ptrConfigPage^.aiFTrigActionPanelRight[5]:=0;
ptrConfigPage^.aiRTrigActionFunctionPanel[1]:=0;
ptrConfigPage^.aiRTrigActionFunctionPanel[2]:=0;
ptrConfigPage^.aiRTrigActionFunctionPanel[3]:=0;
ptrConfigPage^.aiRTrigActionFunctionPanel[4]:=0;
ptrConfigPage^.aiRTrigActionFunctionPanel[5]:=0;
ptrConfigPage^.aiRTrigActionFunctionPanel[6]:=0;
ptrConfigPage^.aiRTrigActionFunctionPanel[7]:=0;
ptrConfigPage^.aiRTrigActionFunctionPanel[8]:=0;
ptrConfigPage^.aiRTrigActionFunctionPanel[9]:=0;
ptrConfigPage^.aiRTrigActionFunctionPanel[10]:=0;
ptrConfigPage^.aiRTrigActionFunctionPanel[11]:=0;
ptrConfigPage^.aiRTrigActionFunctionPanel[12]:=0;
TaskBar_SetupModeB;
ptrConfigPage^.xMaskBtStart:=FALSE;
ptrConfigPage^.xMaskBtStop:=TRUE;
END_ACTION
ACTION TaskBar_BIOS:
(* Navigation panel restriction *)
ptrConfigPage^.aiRTrigActionTouchScreenNavPanel[1,1]:=0;
ptrConfigPage^.aiRTrigActionTouchScreenNavPanel[1,2]:=0;
ptrConfigPage^.aiRTrigActionTouchScreenNavPanel[1,3]:=0;
ptrConfigPage^.aiRTrigActionTouchScreenNavPanel[1,4]:=0;
ptrConfigPage^.aiRTrigActionTouchScreenNavPanel[1,5]:=0;
ptrConfigPage^.aiRTrigActionTouchScreenNavPanel[1,6]:=0;
ptrConfigPage^.aiRTrigActionTouchScreenNavPanel[1,7]:=0;
ptrConfigPage^.aiRTrigActionTouchScreenNavPanel[1,8]:=0;
ptrConfigPage^.aiRTrigActionTouchScreenNavPanel[1,9]:=0;
ptrConfigPage^.aiRTrigActionTouchScreenNavPanel[2,1]:=0;
ptrConfigPage^.aiRTrigActionTouchScreenNavPanel[2,2]:=0;
ptrConfigPage^.aiRTrigActionTouchScreenNavPanel[2,3]:=0;
ptrConfigPage^.aiRTrigActionTouchScreenNavPanel[2,4]:=0;
ptrConfigPage^.aiRTrigActionTouchScreenNavPanel[2,5]:=0;
ptrConfigPage^.aiRTrigActionTouchScreenNavPanel[2,6]:=0;
ptrConfigPage^.aiRTrigActionTouchScreenNavPanel[2,7]:=0;
ptrConfigPage^.aiRTrigActionTouchScreenNavPanel[2,8]:=0;
ptrConfigPage^.aiRTrigActionTouchScreenNavPanel[2,9]:=0;
ptrConfigPage^.aiRTrigActionTouchScreenNavPanel[3,1]:=0;
ptrConfigPage^.aiRTrigActionTouchScreenNavPanel[3,2]:=0;
ptrConfigPage^.aiRTrigActionTouchScreenNavPanel[3,3]:=0;
ptrConfigPage^.aiRTrigActionTouchScreenNavPanel[3,4]:=0;
ptrConfigPage^.aiRTrigActionTouchScreenNavPanel[3,5]:=0;
ptrConfigPage^.aiRTrigActionTouchScreenNavPanel[3,6]:=0;
ptrConfigPage^.aiRTrigActionTouchScreenNavPanel[3,7]:=0;
ptrConfigPage^.aiRTrigActionTouchScreenNavPanel[3,8]:=0;
ptrConfigPage^.aiRTrigActionTouchScreenNavPanel[3,9]:=0;
ptrConfigPage^.aiRTrigActionTouchScreenNavPanel[4,1]:=0;
ptrConfigPage^.aiRTrigActionTouchScreenNavPanel[4,2]:=0;
ptrConfigPage^.aiRTrigActionTouchScreenNavPanel[4,3]:=0;
ptrConfigPage^.aiRTrigActionTouchScreenNavPanel[4,4]:=0;
ptrConfigPage^.aiRTrigActionTouchScreenNavPanel[4,5]:=0;
ptrConfigPage^.aiRTrigActionTouchScreenNavPanel[4,6]:=0;
ptrConfigPage^.aiRTrigActionTouchScreenNavPanel[4,7]:=0;
ptrConfigPage^.aiRTrigActionTouchScreenNavPanel[4,8]:=0;
ptrConfigPage^.aiRTrigActionTouchScreenNavPanel[4,9]:=0;
ptrConfigPage^.aiRTrigActionTouchScreenNavPanel[5,1]:=0;
ptrConfigPage^.aiRTrigActionTouchScreenNavPanel[5,2]:=0;
ptrConfigPage^.aiRTrigActionTouchScreenNavPanel[5,3]:=0;
ptrConfigPage^.aiRTrigActionTouchScreenNavPanel[5,4]:=0;
ptrConfigPage^.aiRTrigActionTouchScreenNavPanel[5,5]:=0;
ptrConfigPage^.aiRTrigActionTouchScreenNavPanel[5,6]:=0;
ptrConfigPage^.aiRTrigActionTouchScreenNavPanel[5,7]:=0;
ptrConfigPage^.aiRTrigActionTouchScreenNavPanel[5,8]:=0;
ptrConfigPage^.aiRTrigActionTouchScreenNavPanel[5,9]:=0;
ptrConfigPage^.aiRTrigActionTouchScreenNavPanel[6,1]:=0;
ptrConfigPage^.aiRTrigActionTouchScreenNavPanel[6,2]:=0;
ptrConfigPage^.aiRTrigActionTouchScreenNavPanel[6,3]:=0;
ptrConfigPage^.aiRTrigActionTouchScreenNavPanel[6,4]:=0;
ptrConfigPage^.aiRTrigActionTouchScreenNavPanel[6,5]:=0;
ptrConfigPage^.aiRTrigActionTouchScreenNavPanel[6,6]:=0;
ptrConfigPage^.aiRTrigActionTouchScreenNavPanel[6,7]:=0;
ptrConfigPage^.aiRTrigActionTouchScreenNavPanel[6,8]:=0;
ptrConfigPage^.aiRTrigActionTouchScreenNavPanel[6,9]:=0;
END_ACTION
ACTION TaskBar_NormalMode:
(* Navigation panel restriction *)
ptrConfigPage^.wMaskTouchScreenNavPanel:=16#3F;
ptrConfigPage^.aiRTrigActionTouchScreenNavPanel[1,1]:=10000 + gT_PageNumber.iAutoMode_Process;
ptrConfigPage^.aiRTrigActionTouchScreenNavPanel[1,2]:=10000 + gT_PageNumber.iAutoMode_ProcessValue1;	(* IGS *)
ptrConfigPage^.aiRTrigActionTouchScreenNavPanel[1,3]:=10000 + gT_PageNumber.iAutoMode_ProcessValue2;	(* IGS *)
ptrConfigPage^.aiRTrigActionTouchScreenNavPanel[1,4]:=10000 + gT_PageNumber.iAutoMode_PartQuality;
ptrConfigPage^.aiRTrigActionTouchScreenNavPanel[1,5]:=0;
ptrConfigPage^.aiRTrigActionTouchScreenNavPanel[1,6]:=0;
ptrConfigPage^.aiRTrigActionTouchScreenNavPanel[1,7]:=0;
ptrConfigPage^.aiRTrigActionTouchScreenNavPanel[1,8]:=0;
ptrConfigPage^.aiRTrigActionTouchScreenNavPanel[1,9]:=0;
ptrConfigPage^.aiRTrigActionTouchScreenNavPanel[2,1]:=10000 + gT_PageNumber.iAutoMode_Referencing;
ptrConfigPage^.aiRTrigActionTouchScreenNavPanel[2,2]:=0;
ptrConfigPage^.aiRTrigActionTouchScreenNavPanel[2,3]:=0;
ptrConfigPage^.aiRTrigActionTouchScreenNavPanel[2,4]:=0;
ptrConfigPage^.aiRTrigActionTouchScreenNavPanel[2,5]:=0;
ptrConfigPage^.aiRTrigActionTouchScreenNavPanel[2,6]:=0;
ptrConfigPage^.aiRTrigActionTouchScreenNavPanel[2,7]:=0;
ptrConfigPage^.aiRTrigActionTouchScreenNavPanel[2,8]:=0;
ptrConfigPage^.aiRTrigActionTouchScreenNavPanel[2,9]:=0;
ptrConfigPage^.aiRTrigActionTouchScreenNavPanel[3,1]:=10000 + gT_PageNumber.iAutoMode_Profile;
ptrConfigPage^.aiRTrigActionTouchScreenNavPanel[3,2]:=0;
ptrConfigPage^.aiRTrigActionTouchScreenNavPanel[3,3]:=0;
ptrConfigPage^.aiRTrigActionTouchScreenNavPanel[3,4]:=0;
ptrConfigPage^.aiRTrigActionTouchScreenNavPanel[3,5]:=0;
ptrConfigPage^.aiRTrigActionTouchScreenNavPanel[3,6]:=0;
ptrConfigPage^.aiRTrigActionTouchScreenNavPanel[3,7]:=0;
ptrConfigPage^.aiRTrigActionTouchScreenNavPanel[3,8]:=0;
ptrConfigPage^.aiRTrigActionTouchScreenNavPanel[3,9]:=0;
ptrConfigPage^.aiRTrigActionTouchScreenNavPanel[4,1]:=10000 + gT_PageNumber.iAutoMode_ToolChange;
ptrConfigPage^.aiRTrigActionTouchScreenNavPanel[4,2]:=10000 + gT_PageNumber.iAutoMode_UserLevel;
ptrConfigPage^.aiRTrigActionTouchScreenNavPanel[4,3]:=10000 + gT_PageNumber.iAutoMode_Language;
ptrConfigPage^.aiRTrigActionTouchScreenNavPanel[4,4]:=0;
ptrConfigPage^.aiRTrigActionTouchScreenNavPanel[4,5]:=0;
ptrConfigPage^.aiRTrigActionTouchScreenNavPanel[4,6]:=0;
ptrConfigPage^.aiRTrigActionTouchScreenNavPanel[4,7]:=0;
ptrConfigPage^.aiRTrigActionTouchScreenNavPanel[4,8]:=0;
ptrConfigPage^.aiRTrigActionTouchScreenNavPanel[4,9]:=0;
ptrConfigPage^.aiRTrigActionTouchScreenNavPanel[5,1]:=10000 + gT_PageNumber.iAutoMode_WPCounter;
ptrConfigPage^.aiRTrigActionTouchScreenNavPanel[5,2]:=10000 + gT_PageNumber.iAutoMode_LampTest;
ptrConfigPage^.aiRTrigActionTouchScreenNavPanel[5,3]:=10000 + gT_PageNumber.iAutoMode_WPCounter;
ptrConfigPage^.aiRTrigActionTouchScreenNavPanel[5,4]:=10000 + gT_PageNumber.iAutoMode_SysInfo;
ptrConfigPage^.aiRTrigActionTouchScreenNavPanel[5,5]:=0;
ptrConfigPage^.aiRTrigActionTouchScreenNavPanel[5,6]:=0;
ptrConfigPage^.aiRTrigActionTouchScreenNavPanel[5,7]:=0;
ptrConfigPage^.aiRTrigActionTouchScreenNavPanel[5,8]:=0;
ptrConfigPage^.aiRTrigActionTouchScreenNavPanel[5,9]:=0;
ptrConfigPage^.aiRTrigActionTouchScreenNavPanel[6,1]:=10000 + gT_PageNumber.iAutoMode_ErrorList;
ptrConfigPage^.aiRTrigActionTouchScreenNavPanel[6,2]:=0;
ptrConfigPage^.aiRTrigActionTouchScreenNavPanel[6,3]:=0;
ptrConfigPage^.aiRTrigActionTouchScreenNavPanel[6,4]:=0;
ptrConfigPage^.aiRTrigActionTouchScreenNavPanel[6,5]:=0;
ptrConfigPage^.aiRTrigActionTouchScreenNavPanel[6,6]:=0;
ptrConfigPage^.aiRTrigActionTouchScreenNavPanel[6,7]:=0;
ptrConfigPage^.aiRTrigActionTouchScreenNavPanel[6,8]:=0;
ptrConfigPage^.aiRTrigActionTouchScreenNavPanel[6,9]:=0;
END_ACTION
ACTION TaskBar_SetupModeA:
(* Navigation panel restriction *)
ptrConfigPage^.wMaskTouchScreenNavPanel:=16#33;
ptrConfigPage^.aiRTrigActionTouchScreenNavPanel[1,1]:=10000 + gT_PageNumber.iHandMode_Process;
ptrConfigPage^.aiRTrigActionTouchScreenNavPanel[1,2]:=10000 + gT_PageNumber.iHandMode_WorkParameter;
ptrConfigPage^.aiRTrigActionTouchScreenNavPanel[1,3]:=10000 + gT_PageNumber.iHandMode_RegulatorPara;
ptrConfigPage^.aiRTrigActionTouchScreenNavPanel[1,4]:=10000 + gT_PageNumber.iHandMode_OnlineChange;
ptrConfigPage^.aiRTrigActionTouchScreenNavPanel[1,5]:=10000 + gT_PageNumber.iHandMode_ConfigPosition;
ptrConfigPage^.aiRTrigActionTouchScreenNavPanel[1,6]:=0;
ptrConfigPage^.aiRTrigActionTouchScreenNavPanel[1,7]:=0;
ptrConfigPage^.aiRTrigActionTouchScreenNavPanel[1,8]:=0;
ptrConfigPage^.aiRTrigActionTouchScreenNavPanel[1,9]:=0;
ptrConfigPage^.aiRTrigActionTouchScreenNavPanel[2,1]:=10000 + gT_PageNumber.iHandMode_ProfileMngmt1;
ptrConfigPage^.aiRTrigActionTouchScreenNavPanel[2,2]:=0;
ptrConfigPage^.aiRTrigActionTouchScreenNavPanel[2,3]:=0;
ptrConfigPage^.aiRTrigActionTouchScreenNavPanel[2,4]:=0;
ptrConfigPage^.aiRTrigActionTouchScreenNavPanel[2,5]:=0;
ptrConfigPage^.aiRTrigActionTouchScreenNavPanel[2,6]:=0;
ptrConfigPage^.aiRTrigActionTouchScreenNavPanel[2,7]:=0;
ptrConfigPage^.aiRTrigActionTouchScreenNavPanel[2,8]:=0;
ptrConfigPage^.aiRTrigActionTouchScreenNavPanel[2,9]:=0;
ptrConfigPage^.aiRTrigActionTouchScreenNavPanel[3,1]:=0;
ptrConfigPage^.aiRTrigActionTouchScreenNavPanel[3,2]:=0;
ptrConfigPage^.aiRTrigActionTouchScreenNavPanel[3,3]:=0;
ptrConfigPage^.aiRTrigActionTouchScreenNavPanel[3,4]:=0;
ptrConfigPage^.aiRTrigActionTouchScreenNavPanel[3,5]:=0;
ptrConfigPage^.aiRTrigActionTouchScreenNavPanel[3,6]:=0;
ptrConfigPage^.aiRTrigActionTouchScreenNavPanel[3,7]:=0;
ptrConfigPage^.aiRTrigActionTouchScreenNavPanel[3,8]:=0;
ptrConfigPage^.aiRTrigActionTouchScreenNavPanel[3,9]:=0;
ptrConfigPage^.aiRTrigActionTouchScreenNavPanel[4,1]:=0;
ptrConfigPage^.aiRTrigActionTouchScreenNavPanel[4,2]:=0;
ptrConfigPage^.aiRTrigActionTouchScreenNavPanel[4,3]:=0;
ptrConfigPage^.aiRTrigActionTouchScreenNavPanel[4,4]:=0;
ptrConfigPage^.aiRTrigActionTouchScreenNavPanel[4,5]:=0;
ptrConfigPage^.aiRTrigActionTouchScreenNavPanel[4,6]:=0;
ptrConfigPage^.aiRTrigActionTouchScreenNavPanel[4,7]:=0;
ptrConfigPage^.aiRTrigActionTouchScreenNavPanel[4,8]:=0;
ptrConfigPage^.aiRTrigActionTouchScreenNavPanel[4,9]:=0;
ptrConfigPage^.aiRTrigActionTouchScreenNavPanel[5,1]:=10000 + gT_PageNumber.iHandMode_Setup1;
ptrConfigPage^.aiRTrigActionTouchScreenNavPanel[5,2]:=0;
ptrConfigPage^.aiRTrigActionTouchScreenNavPanel[5,3]:=0;
ptrConfigPage^.aiRTrigActionTouchScreenNavPanel[5,4]:=0;
ptrConfigPage^.aiRTrigActionTouchScreenNavPanel[5,5]:=0;
ptrConfigPage^.aiRTrigActionTouchScreenNavPanel[5,6]:=0;
ptrConfigPage^.aiRTrigActionTouchScreenNavPanel[5,7]:=0;
ptrConfigPage^.aiRTrigActionTouchScreenNavPanel[5,8]:=0;
ptrConfigPage^.aiRTrigActionTouchScreenNavPanel[5,9]:=0;
ptrConfigPage^.aiRTrigActionTouchScreenNavPanel[6,1]:=10000 + gT_PageNumber.iHandMode_ErrorList;
ptrConfigPage^.aiRTrigActionTouchScreenNavPanel[6,2]:=0;
ptrConfigPage^.aiRTrigActionTouchScreenNavPanel[6,3]:=0;
ptrConfigPage^.aiRTrigActionTouchScreenNavPanel[6,4]:=0;
ptrConfigPage^.aiRTrigActionTouchScreenNavPanel[6,5]:=0;
ptrConfigPage^.aiRTrigActionTouchScreenNavPanel[6,6]:=0;
ptrConfigPage^.aiRTrigActionTouchScreenNavPanel[6,7]:=0;
ptrConfigPage^.aiRTrigActionTouchScreenNavPanel[6,8]:=0;
ptrConfigPage^.aiRTrigActionTouchScreenNavPanel[6,9]:=0;
END_ACTION
ACTION TaskBar_SetupModeB:
(* Navigation panel restriction *)
ptrConfigPage^.wMaskTouchScreenNavPanel:=16#3F;
ptrConfigPage^.aiRTrigActionTouchScreenNavPanel[1,1]:=10000 + gT_PageNumber.iWorkStation_Axis1;
ptrConfigPage^.aiRTrigActionTouchScreenNavPanel[1,2]:=0;;
ptrConfigPage^.aiRTrigActionTouchScreenNavPanel[1,3]:=0;
ptrConfigPage^.aiRTrigActionTouchScreenNavPanel[1,4]:=0;
ptrConfigPage^.aiRTrigActionTouchScreenNavPanel[1,5]:=0;
ptrConfigPage^.aiRTrigActionTouchScreenNavPanel[1,6]:=0;
ptrConfigPage^.aiRTrigActionTouchScreenNavPanel[1,7]:=0;
ptrConfigPage^.aiRTrigActionTouchScreenNavPanel[1,8]:=0;
ptrConfigPage^.aiRTrigActionTouchScreenNavPanel[1,9]:=0;
ptrConfigPage^.aiRTrigActionTouchScreenNavPanel[2,1]:=10000 + gT_PageNumber.iWorkStation_Cylinder1;
ptrConfigPage^.aiRTrigActionTouchScreenNavPanel[2,2]:=0;
ptrConfigPage^.aiRTrigActionTouchScreenNavPanel[2,3]:=0;
ptrConfigPage^.aiRTrigActionTouchScreenNavPanel[2,4]:=0;
ptrConfigPage^.aiRTrigActionTouchScreenNavPanel[2,5]:=0;
ptrConfigPage^.aiRTrigActionTouchScreenNavPanel[2,6]:=0;
ptrConfigPage^.aiRTrigActionTouchScreenNavPanel[2,7]:=0;
ptrConfigPage^.aiRTrigActionTouchScreenNavPanel[2,8]:=0;
ptrConfigPage^.aiRTrigActionTouchScreenNavPanel[2,9]:=0;
ptrConfigPage^.aiRTrigActionTouchScreenNavPanel[3,1]:=10000 + gT_PageNumber.iWorkStation_Valve1;
ptrConfigPage^.aiRTrigActionTouchScreenNavPanel[3,2]:=0;
ptrConfigPage^.aiRTrigActionTouchScreenNavPanel[3,3]:=0;
ptrConfigPage^.aiRTrigActionTouchScreenNavPanel[3,4]:=0;
ptrConfigPage^.aiRTrigActionTouchScreenNavPanel[3,5]:=0;
ptrConfigPage^.aiRTrigActionTouchScreenNavPanel[3,6]:=0;
ptrConfigPage^.aiRTrigActionTouchScreenNavPanel[3,7]:=0;
ptrConfigPage^.aiRTrigActionTouchScreenNavPanel[3,8]:=0;
ptrConfigPage^.aiRTrigActionTouchScreenNavPanel[3,9]:=0;
ptrConfigPage^.aiRTrigActionTouchScreenNavPanel[4,1]:=10000 + gT_PageNumber.iWorkStation_Function1;
ptrConfigPage^.aiRTrigActionTouchScreenNavPanel[4,2]:=0;
ptrConfigPage^.aiRTrigActionTouchScreenNavPanel[4,3]:=0;
ptrConfigPage^.aiRTrigActionTouchScreenNavPanel[4,4]:=0;
ptrConfigPage^.aiRTrigActionTouchScreenNavPanel[4,5]:=0;
ptrConfigPage^.aiRTrigActionTouchScreenNavPanel[4,6]:=0;
ptrConfigPage^.aiRTrigActionTouchScreenNavPanel[4,7]:=0;
ptrConfigPage^.aiRTrigActionTouchScreenNavPanel[4,8]:=0;
ptrConfigPage^.aiRTrigActionTouchScreenNavPanel[4,9]:=0;
ptrConfigPage^.aiRTrigActionTouchScreenNavPanel[5,1]:=10000 + gT_PageNumber.iWorkStation_Setup1;
ptrConfigPage^.aiRTrigActionTouchScreenNavPanel[5,2]:=10000 + gT_PageNumber.iWorkStation_Setup2;
ptrConfigPage^.aiRTrigActionTouchScreenNavPanel[5,3]:=10000 + gT_PageNumber.iWorkStation_Setup3;
ptrConfigPage^.aiRTrigActionTouchScreenNavPanel[5,4]:=10000 + gT_PageNumber.iWorkStation_Setup4;
ptrConfigPage^.aiRTrigActionTouchScreenNavPanel[5,5]:=10000 + gT_PageNumber.iWorkStation_Setup5;
ptrConfigPage^.aiRTrigActionTouchScreenNavPanel[5,6]:=0;
ptrConfigPage^.aiRTrigActionTouchScreenNavPanel[5,7]:=0;
ptrConfigPage^.aiRTrigActionTouchScreenNavPanel[5,8]:=0;
ptrConfigPage^.aiRTrigActionTouchScreenNavPanel[5,9]:=0;
ptrConfigPage^.aiRTrigActionTouchScreenNavPanel[6,1]:=10000 + gT_PageNumber.iWorkStation_ErrorList;
ptrConfigPage^.aiRTrigActionTouchScreenNavPanel[6,2]:=0;
ptrConfigPage^.aiRTrigActionTouchScreenNavPanel[6,3]:=0;
ptrConfigPage^.aiRTrigActionTouchScreenNavPanel[6,4]:=0;
ptrConfigPage^.aiRTrigActionTouchScreenNavPanel[6,5]:=0;
ptrConfigPage^.aiRTrigActionTouchScreenNavPanel[6,6]:=0;
ptrConfigPage^.aiRTrigActionTouchScreenNavPanel[6,7]:=0;
ptrConfigPage^.aiRTrigActionTouchScreenNavPanel[6,8]:=0;
ptrConfigPage^.aiRTrigActionTouchScreenNavPanel[6,9]:=0;
END_ACTION

(* POU GENERAL/PROFILE/FB_COMPAREPROFILEPROCESSVALUE, ST *)
FUNCTION_BLOCK FB_COMPAREPROFILEPROCESSVALUE
VAR_INPUT
	T_LoadProfileParameter:ST_RETAIN_DATA_PROFILEPARAMETER;	(* Profil Parameter für Profil(LoadData) *)
	T_ProfileParameter:ST_RETAIN_DATA_PROFILEPARAMETER;	(* Profil Parameter für Profil(Data) *)
END_VAR
VAR_OUTPUT
	xProcessValueModified:BOOL;
END_VAR
VAR_IN_OUT
END_VAR
VAR
(* variable *)
	rTmpDifference: REAL;
	rTolerance:REAL:=0.001;
END_VAR
(* compare value *)
	xProcessValueModified:=FALSE;
	(* value *)
	IF T_LoadProfileParameter.T_ProfileOnlineChange.rTorqueLevelHC <> T_ProfileParameter.T_ProfileOnlineChange.rTorqueLevelHC THEN
		rTmpDifference:=ABS(T_LoadProfileParameter.T_ProfileOnlineChange.rTorqueLevelHC - T_ProfileParameter.T_ProfileOnlineChange.rTorqueLevelHC);
		IF (rTmpDifference > rTolerance) THEN
			xProcessValueModified:=TRUE;
		END_IF;
	END_IF
	IF T_LoadProfileParameter.T_ProfileOnlineChange.rForceDeflection <> T_ProfileParameter.T_ProfileOnlineChange.rForceDeflection THEN
		rTmpDifference:=ABS(T_LoadProfileParameter.T_ProfileOnlineChange.rForceDeflection - T_ProfileParameter.T_ProfileOnlineChange.rForceDeflection);
		IF (rTmpDifference > rTolerance) THEN
			xProcessValueModified:=TRUE;
		END_IF;
	END_IF
	IF T_LoadProfileParameter.T_ProfileOnlineChange.rWorkingSpeedForward <> T_ProfileParameter.T_ProfileOnlineChange.rWorkingSpeedForward THEN
		rTmpDifference:=ABS(T_LoadProfileParameter.T_ProfileOnlineChange.rWorkingSpeedForward - T_ProfileParameter.T_ProfileOnlineChange.rWorkingSpeedForward);
		IF (rTmpDifference > rTolerance) THEN
			xProcessValueModified:=TRUE;
		END_IF;
	END_IF
	IF T_LoadProfileParameter.T_ProfileOnlineChange.rWorkingOffsetBackward <> T_ProfileParameter.T_ProfileOnlineChange.rWorkingOffsetBackward THEN
		rTmpDifference:=ABS(T_LoadProfileParameter.T_ProfileOnlineChange.rWorkingOffsetBackward - T_ProfileParameter.T_ProfileOnlineChange.rWorkingOffsetBackward);
		IF (rTmpDifference > rTolerance) THEN
			xProcessValueModified:=TRUE;
		END_IF;
	END_IF
	IF T_LoadProfileParameter.T_ProfileOnlineChange.rWorkingSpeedBackward <> T_ProfileParameter.T_ProfileOnlineChange.rWorkingSpeedBackward THEN
		rTmpDifference:=ABS(T_LoadProfileParameter.T_ProfileOnlineChange.rWorkingSpeedBackward - T_ProfileParameter.T_ProfileOnlineChange.rWorkingSpeedBackward);
		IF (rTmpDifference > rTolerance) THEN
			xProcessValueModified:=TRUE;
		END_IF;
	END_IF
	IF T_LoadProfileParameter.T_ProfileOnlineChange.rWorkingSpindleSpeed <> T_ProfileParameter.T_ProfileOnlineChange.rWorkingSpindleSpeed THEN
		rTmpDifference:=ABS(T_LoadProfileParameter.T_ProfileOnlineChange.rWorkingSpindleSpeed - T_ProfileParameter.T_ProfileOnlineChange.rWorkingSpindleSpeed);
		IF (rTmpDifference > rTolerance) THEN
			xProcessValueModified:=TRUE;
		END_IF;
	END_IF

	IF T_LoadProfileParameter.T_ProzessData.rPositionLoad <> T_ProfileParameter.T_ProzessData.rPositionLoad THEN xProcessValueModified:=TRUE; END_IF
	IF T_LoadProfileParameter.T_ProzessData.rPositionStartProc <> T_ProfileParameter.T_ProzessData.rPositionStartProc THEN xProcessValueModified:=TRUE; END_IF
	IF T_LoadProfileParameter.T_ProzessData.rPositionEndProc <> T_ProfileParameter.T_ProzessData.rPositionEndProc THEN xProcessValueModified:=TRUE; END_IF
	IF T_LoadProfileParameter.T_ProzessData.rPositionToolChange <> T_ProfileParameter.T_ProzessData.rPositionToolChange THEN xProcessValueModified:=TRUE; END_IF
	IF T_LoadProfileParameter.T_ProzessData.rInfeedZAxisSpeed <> T_ProfileParameter.T_ProzessData.rInfeedZAxisSpeed THEN xProcessValueModified:=TRUE; END_IF
	IF T_LoadProfileParameter.T_ProzessData.rInfeedSpindleSpeed <> T_ProfileParameter.T_ProzessData.rInfeedSpindleSpeed THEN xProcessValueModified:=TRUE; END_IF
	IF T_LoadProfileParameter.T_ProzessData.rOutfeedStrokeAxisSpeed <> T_ProfileParameter.T_ProzessData.rOutfeedStrokeAxisSpeed THEN xProcessValueModified:=TRUE; END_IF
	IF T_LoadProfileParameter.T_ProzessData.rOutfeedSpindleSpeed <> T_ProfileParameter.T_ProzessData.rOutfeedSpindleSpeed THEN xProcessValueModified:=TRUE; END_IF
	IF T_LoadProfileParameter.T_ProzessData.rInfeedForceDeflection <> T_ProfileParameter.T_ProzessData.rInfeedForceDeflection THEN xProcessValueModified:=TRUE; END_IF
	IF T_LoadProfileParameter.T_ProzessData.rInfeedOffsetBackward <> T_ProfileParameter.T_ProzessData.rInfeedOffsetBackward THEN xProcessValueModified:=TRUE; END_IF
	IF T_LoadProfileParameter.T_ProzessData.iNumberTryInfeed <> T_ProfileParameter.T_ProzessData.iNumberTryInfeed THEN xProcessValueModified:=TRUE; END_IF

	IF T_LoadProfileParameter.T_ProzessData.rProcessMinTime <> T_ProfileParameter.T_ProzessData.rProcessMinTime THEN xProcessValueModified:=TRUE; END_IF
	IF T_LoadProfileParameter.T_ProzessData.rProcessMaxTime <> T_ProfileParameter.T_ProzessData.rProcessMaxTime THEN xProcessValueModified:=TRUE; END_IF
	IF T_LoadProfileParameter.T_ProzessData.iHCStartProcPosCounter <> T_ProfileParameter.T_ProzessData.iHCStartProcPosCounter THEN xProcessValueModified:=TRUE; END_IF
	IF T_LoadProfileParameter.T_ProzessData.rDeflectionSensorOffset <> T_ProfileParameter.T_ProzessData.rDeflectionSensorOffset THEN xProcessValueModified:=TRUE; END_IF
	IF T_LoadProfileParameter.T_ProzessData.rTorqueLevel_Overload <> T_ProfileParameter.T_ProzessData.rTorqueLevel_Overload THEN xProcessValueModified:=TRUE; END_IF

	IF T_LoadProfileParameter.T_ProzessData.iSparkOutStrokeCount <> T_ProfileParameter.T_ProzessData.iSparkOutStrokeCount THEN xProcessValueModified:=TRUE; END_IF
	IF T_LoadProfileParameter.T_ProzessData.rSparkOutStrokeLength <> T_ProfileParameter.T_ProzessData.rSparkOutStrokeLength THEN xProcessValueModified:=TRUE; END_IF
	IF T_LoadProfileParameter.T_ProzessData.rSparkOutStrokeSpeed <> T_ProfileParameter.T_ProzessData.rSparkOutStrokeSpeed THEN xProcessValueModified:=TRUE; END_IF
	IF T_LoadProfileParameter.T_ProzessData.rSparkOutForceDeflection <> T_ProfileParameter.T_ProzessData.rSparkOutForceDeflection THEN xProcessValueModified:=TRUE; END_IF
	IF T_LoadProfileParameter.T_ProzessData.rSparkOutTorqueLevel <> T_ProfileParameter.T_ProzessData.rSparkOutTorqueLevel THEN xProcessValueModified:=TRUE; END_IF

	IF T_LoadProfileParameter.T_ProzessData.rPosToolGuid_Up <> T_ProfileParameter.T_ProzessData.rPosToolGuid_Up THEN xProcessValueModified:=TRUE; END_IF
	IF T_LoadProfileParameter.T_ProzessData.rPosToolGuid_Down <> T_ProfileParameter.T_ProzessData.rPosToolGuid_Down THEN xProcessValueModified:=TRUE; END_IF
	IF T_LoadProfileParameter.T_ProzessData.rDistanceToolGuide <> T_ProfileParameter.T_ProzessData.rDistanceToolGuide THEN xProcessValueModified:=TRUE; END_IF
	IF T_LoadProfileParameter.T_ProzessData.rDistanceToolEndPos <> T_ProfileParameter.T_ProzessData.rDistanceToolEndPos THEN xProcessValueModified:=TRUE; END_IF
	IF T_LoadProfileParameter.T_ProzessData.rLengthTool_Fixed <> T_ProfileParameter.T_ProzessData.rLengthTool_Fixed THEN xProcessValueModified:=TRUE; END_IF
	IF T_LoadProfileParameter.T_ProzessData.rLengthTool_Work <> T_ProfileParameter.T_ProzessData.rLengthTool_Work THEN xProcessValueModified:=TRUE; END_IF
	IF T_LoadProfileParameter.T_ProzessData.rLengthToolGuide <> T_ProfileParameter.T_ProzessData.rLengthToolGuide THEN xProcessValueModified:=TRUE; END_IF
	IF T_LoadProfileParameter.T_ProzessData.rLengthAirTableBoard <> T_ProfileParameter.T_ProzessData.rLengthAirTableBoard THEN xProcessValueModified:=TRUE; END_IF
	IF T_LoadProfileParameter.T_ProzessData.xConfigActive <> T_ProfileParameter.T_ProzessData.xConfigActive THEN xProcessValueModified:=TRUE; END_IF

	IF T_LoadProfileParameter.T_ProzessData.iMaxTorque <> T_ProfileParameter.T_ProzessData.iMaxTorque THEN xProcessValueModified:=TRUE; END_IF
	IF T_LoadProfileParameter.T_ProzessData.rSpeedZAxisForBackward <> T_ProfileParameter.T_ProzessData.rSpeedZAxisForBackward THEN xProcessValueModified:=TRUE; END_IF
	IF T_LoadProfileParameter.T_ProzessData.rWorkingSpeedOscillation <> T_ProfileParameter.T_ProzessData.rWorkingSpeedOscillation THEN xProcessValueModified:=TRUE; END_IF
	IF T_LoadProfileParameter.T_ProzessData.rZ1AxisPosSwitchOAxisOff <> T_ProfileParameter.T_ProzessData.rZ1AxisPosSwitchOAxisOff THEN xProcessValueModified:=TRUE; END_IF
	IF T_LoadProfileParameter.T_ProzessData.xActivateCoolantProcess <> T_ProfileParameter.T_ProzessData.xActivateCoolantProcess THEN xProcessValueModified:=TRUE; END_IF
	IF T_LoadProfileParameter.T_ProzessData.rStrokeAxisPosSwitchCoolantOff <> T_ProfileParameter.T_ProzessData.rStrokeAxisPosSwitchCoolantOff THEN xProcessValueModified:=TRUE; END_IF

	IF T_LoadProfileParameter.T_ProzessData.rCentringPosZ1Axis <> T_ProfileParameter.T_ProzessData.rCentringPosZ1Axis THEN xProcessValueModified:=TRUE; END_IF
	IF T_LoadProfileParameter.T_ProzessData.rCentringPosSpeedSlowZ1Axis <> T_ProfileParameter.T_ProzessData.rCentringPosSpeedSlowZ1Axis THEN xProcessValueModified:=TRUE; END_IF
	IF T_LoadProfileParameter.T_ProzessData.rCentringPosSpeedFastZ1Axis <> T_ProfileParameter.T_ProzessData.rCentringPosSpeedFastZ1Axis THEN xProcessValueModified:=TRUE; END_IF
	IF T_LoadProfileParameter.T_ProzessData.rCentringSpeedSAxis <> T_ProfileParameter.T_ProzessData.rCentringSpeedSAxis THEN xProcessValueModified:=TRUE; END_IF
	IF T_LoadProfileParameter.T_ProzessData.rCentringSpeedOAxis <> T_ProfileParameter.T_ProzessData.rCentringSpeedOAxis THEN xProcessValueModified:=TRUE; END_IF
	IF T_LoadProfileParameter.T_ProzessData.rCentringBackStrokeOffsetFirstHC <> T_ProfileParameter.T_ProzessData.rCentringBackStrokeOffsetFirstHC THEN xProcessValueModified:=TRUE; END_IF
	IF T_LoadProfileParameter.T_ProzessData.rCentringBackStrokeOffsetAfterFirstHC <> T_ProfileParameter.T_ProzessData.rCentringBackStrokeOffsetAfterFirstHC THEN xProcessValueModified:=TRUE; END_IF
	IF T_LoadProfileParameter.T_ProzessData.rCentringOffsetBeforeLastHC <> T_ProfileParameter.T_ProzessData.rCentringOffsetBeforeLastHC THEN xProcessValueModified:=TRUE; END_IF
	IF T_LoadProfileParameter.T_ProzessData.rCentringBackStrokeSpeed <> T_ProfileParameter.T_ProzessData.rCentringBackStrokeSpeed THEN xProcessValueModified:=TRUE; END_IF
	IF T_LoadProfileParameter.T_ProzessData.rCentringTimeHCActive <> T_ProfileParameter.T_ProzessData.rCentringTimeHCActive THEN xProcessValueModified:=TRUE; END_IF
	IF T_LoadProfileParameter.T_ProzessData.rCentringTimeHCInactive <> T_ProfileParameter.T_ProzessData.rCentringTimeHCInactive THEN xProcessValueModified:=TRUE; END_IF
	IF T_LoadProfileParameter.T_ProzessData.iCentringNumberMaxHCinWindow <> T_ProfileParameter.T_ProzessData.iCentringNumberMaxHCinWindow THEN xProcessValueModified:=TRUE; END_IF
	IF T_LoadProfileParameter.T_ProzessData.rCentringHCWindow <> T_ProfileParameter.T_ProzessData.rCentringHCWindow THEN xProcessValueModified:=TRUE; END_IF
	IF T_LoadProfileParameter.T_ProzessData.rCentringForceDeflection <> T_ProfileParameter.T_ProzessData.rCentringForceDeflection THEN xProcessValueModified:=TRUE; END_IF
	IF T_LoadProfileParameter.T_ProzessData.rCentringOffsetBackward <> T_ProfileParameter.T_ProzessData.rCentringOffsetBackward THEN xProcessValueModified:=TRUE; END_IF
	IF T_LoadProfileParameter.T_ProzessData.rCenteringDeflectionSensorOffset <> T_ProfileParameter.T_ProzessData.rCenteringDeflectionSensorOffset THEN xProcessValueModified:=TRUE; END_IF
	IF T_LoadProfileParameter.T_ProzessData.rCentringOffsetSlowToFastZSpeed <> T_ProfileParameter.T_ProzessData.rCentringOffsetSlowToFastZSpeed THEN xProcessValueModified:=TRUE; END_IF
	IF T_LoadProfileParameter.T_ProzessData.iCentringSelectProcess <> T_ProfileParameter.T_ProzessData.iCentringSelectProcess THEN xProcessValueModified:=TRUE; END_IF
	IF T_LoadProfileParameter.T_ProzessData.xPositionEndProcIncOnOff <> T_ProfileParameter.T_ProzessData.xPositionEndProcIncOnOff THEN xProcessValueModified:=TRUE; END_IF
	IF T_LoadProfileParameter.T_ProzessData.rPositionEndProcMaxInc <> T_ProfileParameter.T_ProzessData.rPositionEndProcMaxInc THEN xProcessValueModified:=TRUE; END_IF
	IF T_LoadProfileParameter.T_ProzessData.rPositionEndProInc <> T_ProfileParameter.T_ProzessData.rPositionEndProInc THEN xProcessValueModified:=TRUE; END_IF
	IF T_LoadProfileParameter.T_ProzessData.rOutfeedStrokeAxisSpeedSlow <> T_ProfileParameter.T_ProzessData.rOutfeedStrokeAxisSpeedSlow THEN xProcessValueModified:=TRUE; END_IF
	IF T_LoadProfileParameter.T_ProzessData.rZ1AxisPosSwitchFastVel <> T_ProfileParameter.T_ProzessData.rZ1AxisPosSwitchFastVel THEN xProcessValueModified:=TRUE; END_IF
	IF T_LoadProfileParameter.T_ProzessData.rZ1AxisOffsetStartRecordTorque <> T_ProfileParameter.T_ProzessData.rZ1AxisOffsetStartRecordTorque THEN xProcessValueModified:=TRUE; END_IF
	IF T_LoadProfileParameter.T_ProzessData.xCentringEndProcIncOnOff <> T_ProfileParameter.T_ProzessData.xCentringEndProcIncOnOff THEN xProcessValueModified:=TRUE; END_IF
	IF T_LoadProfileParameter.T_ProzessData.rCentringEndProInc <> T_ProfileParameter.T_ProzessData.rCentringEndProInc THEN xProcessValueModified:=TRUE; END_IF
	IF T_LoadProfileParameter.T_ProzessData.rWorkingSpindleSpeedMinMax <> T_ProfileParameter.T_ProzessData.rWorkingSpindleSpeedMinMax THEN xProcessValueModified:=TRUE; END_IF
	IF T_LoadProfileParameter.T_ProzessData.rO_Ctrl_TorquePercent_OFF <> T_ProfileParameter.T_ProzessData.rO_Ctrl_TorquePercent_OFF THEN xProcessValueModified:=TRUE; END_IF
	IF T_LoadProfileParameter.T_ProzessData.rO_Ctrl_HystereseOffset <> T_ProfileParameter.T_ProzessData.rO_Ctrl_HystereseOffset THEN xProcessValueModified:=TRUE; END_IF
	IF T_LoadProfileParameter.T_ProzessData.rZPositionCylindricalArea <> T_ProfileParameter.T_ProzessData.rZPositionCylindricalArea THEN xProcessValueModified:=TRUE; END_IF
	IF T_LoadProfileParameter.T_ProzessData.rZMinThresholdTroqueEndProcess <> T_ProfileParameter.T_ProzessData.rZMinThresholdTroqueEndProcess THEN xProcessValueModified:=TRUE; END_IF

	IF T_LoadProfileParameter.T_ProzessData.iWorkControlType <> T_ProfileParameter.T_ProzessData.iWorkControlType THEN xProcessValueModified:=TRUE; END_IF
	IF T_LoadProfileParameter.T_ProzessData.rZ_PID_Torque <> T_ProfileParameter.T_ProzessData.rZ_PID_Torque THEN xProcessValueModified:=TRUE; END_IF
	IF T_LoadProfileParameter.T_ProzessData.rZ_PID_MinSpeed <> T_ProfileParameter.T_ProzessData.rZ_PID_MinSpeed THEN xProcessValueModified:=TRUE; END_IF
	IF T_LoadProfileParameter.T_ProzessData.rZ_PID_MaxSpeed <> T_ProfileParameter.T_ProzessData.rZ_PID_MaxSpeed THEN xProcessValueModified:=TRUE; END_IF
	IF T_LoadProfileParameter.T_ProzessData.rZ_PID_Kp <> T_ProfileParameter.T_ProzessData.rZ_PID_Kp THEN xProcessValueModified:=TRUE; END_IF
	IF T_LoadProfileParameter.T_ProzessData.rZ_PID_Ki <> T_ProfileParameter.T_ProzessData.rZ_PID_Ki THEN xProcessValueModified:=TRUE; END_IF
	IF T_LoadProfileParameter.T_ProzessData.rZ_PID_Kd <> T_ProfileParameter.T_ProzessData.rZ_PID_Kd THEN xProcessValueModified:=TRUE; END_IF
	IF T_LoadProfileParameter.T_ProzessData.iZ_PID_FilterM <> T_ProfileParameter.T_ProzessData.iZ_PID_FilterM THEN xProcessValueModified:=TRUE; END_IF
	IF T_LoadProfileParameter.T_ProzessData.rZ_D_Kd <> T_ProfileParameter.T_ProzessData.rZ_D_Kd THEN xProcessValueModified:=TRUE; END_IF
	IF T_LoadProfileParameter.T_ProzessData.iZ_D_FilterM <> T_ProfileParameter.T_ProzessData.iZ_D_FilterM THEN xProcessValueModified:=TRUE; END_IF

	IF T_LoadProfileParameter.T_ProzessData.rSuspensionBubblerSpeed <> T_ProfileParameter.T_ProzessData.rSuspensionBubblerSpeed THEN xProcessValueModified:=TRUE; END_IF
	IF T_LoadProfileParameter.T_ProzessData.rSuspensionFeederSpeed <> T_ProfileParameter.T_ProzessData.rSuspensionFeederSpeed THEN xProcessValueModified:=TRUE; END_IF

	IF T_LoadProfileParameter.T_ProzessData.rDistProgressStroke <> T_ProfileParameter.T_ProzessData.rDistProgressStroke THEN xProcessValueModified:=TRUE; END_IF
	IF T_LoadProfileParameter.T_ProzessData.iProgressStrokeStartTorque <> T_ProfileParameter.T_ProzessData.iProgressStrokeStartTorque THEN xProcessValueModified:=TRUE; END_IF
	IF T_LoadProfileParameter.T_ProzessData.iCleanNozzleMode <> T_ProfileParameter.T_ProzessData.iCleanNozzleMode THEN xProcessValueModified:=TRUE; END_IF
END_FUNCTION_BLOCK

(* POU PRG_LAYER5_VISU/FB_VISU/Function/FB_GetParameterList, ST *)
FUNCTION_BLOCK FB_GetParameterList
VAR_INPUT
	xNormalModeActive:BOOL;
	iSetupMode:INT;
	wActiveTaskBar:WORD;
	iActLevel:INT;
END_VAR
VAR_IN_OUT
	aiTempActiveParaListState:ARRAY [0..3,1..6] OF INT;
END_VAR
VAR_OUTPUT
	iParameterList:INT;
	wNotMasktext:WORD;
	wState:WORD;
	aiSelectText:ARRAY [1..15] OF INT;
	bParameterListEditable:BYTE;
	bMessageParameter:BYTE;		(* 0=Unterdrücken der Parameter Nachricht, 1=Nur mittels Operator Level, 2=Nur mittels System Level, 3=Keine Parameterliste vorhanden *)
END_VAR
VAR
	xInit: BOOL;
	ii: INT;
	jj: INT;
	iTask: INT;
END_VAR
IF NOT(xInit) THEN
	xInit:=TRUE;
	FOR ii:=0 TO 3 DO
		FOR jj:=1 TO 6 DO
			aiTempActiveParaListState[ii,jj]:=1;
		END_FOR;
	END_FOR;
END_IF;
iParameterList:=0;
wNotMasktext:=16#FFF;
aiSelectText[1]:=aiSelectText[2]:=aiSelectText[3]:=aiSelectText[4]:=aiSelectText[5]:=0;
aiSelectText[6]:=aiSelectText[7]:=aiSelectText[8]:=aiSelectText[9]:=aiSelectText[10]:=0;
aiSelectText[11]:=aiSelectText[12]:=aiSelectText[13]:=aiSelectText[14]:=aiSelectText[15]:=0;
wState:=0;
bParameterListEditable:=0;
bMessageParameter:=3;
iTask:=iFct_GetBitNumber(wInputButton:=wActiveTaskBar);
IF xNormalModeActive THEN
	CASE iTask OF
	(* NormalBetrieb -->Task 1,2,3,4,5,6 *)
	1,2,3,4,5,6:	IF (aiTempActiveParaListState[0,iTask] > 3) THEN aiTempActiveParaListState[0,iTask]:=1; END_IF;
				CASE aiTempActiveParaListState[0,iTask] OF
				1:	iParameterList:=10;
					wState:=16#1;			(* Liste 1 ausgewählt *)
				2:	iParameterList:=11;
					wState:=16#2;			(* Liste 2 ausgewählt *)
				3:	iParameterList:=12;
					wState:=16#4;			(* Liste 3 ausgewählt *)
				END_CASE;
				wNotMasktext:=16#FFF8;	(* Liste 1,2,3 darf nicht unterdrückt werden *)
				aiSelectText[1]:=10;
				aiSelectText[2]:=11;
				aiSelectText[3]:=12;
				IF (iActLevel > 0) THEN
					bMessageParameter:=0;
				ELSE
					bMessageParameter:=1;
					iParameterList:=0;
				END_IF;
				bParameterListEditable:=1;	(* Parameterliste Editierbar *)
	END_CASE;
ELSE
	IF (iSetupMode = 1) THEN
		CASE iTask OF
		(* EinrichtBetrieb A-->Task 1,2,3,4,5,6 *)
		1,2,3,4,5,6:	IF (aiTempActiveParaListState[iSetupMode,iTask] > 15) THEN aiTempActiveParaListState[iSetupMode,iTask]:=1; END_IF;
					CASE aiTempActiveParaListState[iSetupMode,iTask] OF
					1:	iParameterList:=110;
						wState:=16#1;			(* Liste 1 ausgewählt *)
					2:	iParameterList:=111;
						wState:=16#2;			(* Liste 2 ausgewählt *)
					3:	iParameterList:=112;
						wState:=16#4;			(* Liste 3 ausgewählt *)
					4:	iParameterList:=113;
						wState:=16#8;			(* Liste 4 ausgewählt *)
					5:	iParameterList:=114;
						wState:=16#10;		(* Liste 5 ausgewählt *)
					6:	iParameterList:=115;
						wState:=16#20;		(* Liste 6 ausgewählt *)
					7:	iParameterList:=116;
						wState:=16#40;		(* Liste 7 ausgewählt *)
					8:	iParameterList:=117;
						wState:=16#80;		(* Liste 8 ausgewählt *)
					15:	iParameterList:=124;
						wState:=16#4000;		(* Liste 15 ausgewählt *)
					END_CASE;
					aiSelectText[1]:=110;
					aiSelectText[2]:=111;
					aiSelectText[3]:=112;
					aiSelectText[4]:=113;
					aiSelectText[5]:=114;
					aiSelectText[6]:=115;
					aiSelectText[7]:=116;
					aiSelectText[8]:=117;
					aiSelectText[15]:=124;
					wNotMasktext:=16#BF00;	(* Liste 1,2,3,4,5,6,15 dürfen nicht unterdrückt werden *)
					bParameterListEditable:=1;	(* Parameterliste Editierbar *)
					bMessageParameter:=0;
		END_CASE;
	ELSIF (iSetupMode = 2) THEN
		CASE iTask OF
		(* EinrichtBetrieb B-->Task 1,2,3,4,5,6 *)
		1,2,3,4,5,6:	IF (aiTempActiveParaListState[iSetupMode,iTask] > 8) THEN aiTempActiveParaListState[iSetupMode,iTask]:=1; END_IF;
					CASE aiTempActiveParaListState[iSetupMode,iTask] OF
					1:	iParameterList:=210;
						wState:=16#1;			(* Liste 1 ausgewählt *)
					2:	iParameterList:=211;
						wState:=16#2;			(* Liste 2 ausgewählt *)
					3:	iParameterList:=212;
						wState:=16#4;			(* Liste 3 ausgewählt *)
					4:	iParameterList:=213;
						wState:=16#8;			(* Liste 4 ausgewählt *)
					5:	iParameterList:=214;
						wState:=16#10;		(* Liste 5 ausgewählt *)
					6:	iParameterList:=215;
						wState:=16#20;		(* Liste 6 ausgewählt *)
					7:	iParameterList:=216;
						wState:=16#40;		(* Liste 7 ausgewählt *)
					8:	iParameterList:=217;
						wState:=16#80;		(* Liste 8 ausgewählt *)
					END_CASE;
					IF (aiTempActiveParaListState[iSetupMode,iTask] = 1) OR (aiTempActiveParaListState[iSetupMode,iTask] = 6) THEN
						bMessageParameter:=0;
					ELSE
						IF (iActLevel > 1) THEN
							bMessageParameter:=0;
						ELSE
							bMessageParameter:=2;	(* Nur mittels System Level *)
							iParameterList:=0;
						END_IF;
					END_IF;
					aiSelectText[1]:=210;
					aiSelectText[2]:=211;
					aiSelectText[3]:=212;
					aiSelectText[4]:=213;
					aiSelectText[5]:=214;
					aiSelectText[6]:=215;
					aiSelectText[7]:=216;
					aiSelectText[8]:=217;
					wNotMasktext:=16#FF00;	(* Liste 1,2,3,4,5,6,7 und 8 dürfen nicht unterdrückt werden *)
					bParameterListEditable:=1;	(* Parameterliste Editierbar *)
		END_CASE;
	END_IF;
END_IF;
END_FUNCTION_BLOCK

(* POU PRG_LAYER5_VISU/FB_VISU/Function/iFct_GetBitNumber, ST *)
FUNCTION iFct_GetBitNumber : INT
VAR_INPUT
	wInputButton:WORD;
END_VAR
VAR
	wTmp:WORD;
	ii: INT;
END_VAR
iFct_GetBitNumber:=0;
wTmp:=wInputButton;
FOR  ii:=1 TO 16 DO	(* Only for datatype WORD-->16Bit *)
	IF (wTmp AND 16#1) = 16#1 THEN
		iFct_GetBitNumber:=ii;	(* Only the first Bit from the right side  will be check-->be sure that it is settled only one bit *)
		EXIT;
	END_IF;
	wTmp:=ROR(wTmp,1);	(* Shift 1 Bit to right *)
END_FOR;
END_FUNCTION

(* POU GENERAL/FB_WRAP_WPQUALITY, ST *)
FUNCTION_BLOCK FB_WRAP_WPQUALITY
VAR_INPUT
	T_PartAnalysis:ST_PARTANALYSIS;
END_VAR
VAR_IN_OUT
	diHoleNumber:DINT;
END_VAR
VAR_OUTPUT
	T_DataOut:ST_PARTANALYSIS_OUTPUT;
END_VAR
VAR
	diTmpHoleNumber: DINT;
	ii:INT;
END_VAR
IF (diHoleNumber <> 0) THEN
	FOR ii:=1 TO ciMaxWP DO
		IF (T_PartAnalysis.adiNumberHole[ii] = diHoleNumber) THEN
			diTmpHoleNumber:=ii;
		END_IF;
	END_FOR;
	IF (diTmpHoleNumber < 1) THEN
		diTmpHoleNumber:=1;
	END_IF;
	IF (diTmpHoleNumber > ciMaxWP) THEN
		diTmpHoleNumber:=ciMaxWP;
	END_IF;
	T_DataOut.bHole_WorkPartQuality:=T_PartAnalysis.abWorkPartQuality[diTmpHoleNumber];
	T_DataOut.diHole_CycleTime:=T_PartAnalysis.adiCycleTime[diTmpHoleNumber];
	T_DataOut.diHole_WorkTime:=T_PartAnalysis.adiWorkTime[diTmpHoleNumber];
	T_DataOut.iHole_HCCounter:=T_PartAnalysis.aiHCCounter[diTmpHoleNumber];
	T_DataOut.iHole_HCCounterCentering:=T_PartAnalysis.aiHCCounterCentering[diTmpHoleNumber];
	T_DataOut.iHole_HCCounterTorque:=T_PartAnalysis.aiHCCounterTorque[diTmpHoleNumber];
	T_DataOut.iHole_HCCounterSpeed:=T_PartAnalysis.aiHCCounterSpeed[diTmpHoleNumber];
	T_DataOut.rHole_FirstHC:=T_PartAnalysis.arFirstHC[diTmpHoleNumber];
	T_DataOut.bHole_InfeedCounterZ:=T_PartAnalysis.abInfeedCounterZ[diTmpHoleNumber];
ELSE
	T_DataOut.bHole_WorkPartQuality:=0;
	T_DataOut.diHole_CycleTime:=0;
	T_DataOut.diHole_WorkTime:=0;
	T_DataOut.iHole_HCCounter:=0;
	T_DataOut.iHole_HCCounterCentering:=0;
	T_DataOut.iHole_HCCounterTorque:=0;
	T_DataOut.iHole_HCCounterSpeed:=0;
	T_DataOut.rHole_FirstHC:=0.0;
	T_DataOut.bHole_InfeedCounterZ:=0;
END_IF;
END_FUNCTION_BLOCK

(* POU GENERAL/FB_Linearization_Potentiometer, ST *)
FUNCTION_BLOCK FB_Linearization_Potentiometer
VAR_INPUT
	adi_X_MeasurePoint_Voltage:ARRAY [0..11] OF DINT;	(* 0 - 32768 *)
	lr_X_Voltage:LREAL;	(* 0 - 32768 *)
END_VAR
VAR_OUTPUT
	lrValuePercent:LREAL;		(* in N *)
	lrScaledValuePercent:LREAL;	(* in N *)
END_VAR
VAR
	ii: INT;
	lr_M_gradient: LREAL;
	lr_B_AxisIntercept: LREAL;
	adi_X_FixedValue:ARRAY [0..10] OF DINT;
END_VAR
(***********************************               Linearisierung für Potentiometer              ***********************************)
lr_M_gradient:=0.0;
lr_B_AxisIntercept:=0.0;
lrValuePercent:=lrScaledValuePercent:=0.0;
adi_X_FixedValue[0]:=0;
adi_X_FixedValue[1]:=10;
adi_X_FixedValue[2]:=20;
adi_X_FixedValue[3]:=30;
adi_X_FixedValue[4]:=40;
adi_X_FixedValue[5]:=50;
adi_X_FixedValue[6]:=60;
adi_X_FixedValue[7]:=70;
adi_X_FixedValue[8]:=80;
adi_X_FixedValue[9]:=90;
adi_X_FixedValue[10]:=100;
IF (lr_X_Voltage <> 0) THEN
	FOR ii:=0 TO 9 DO
		IF (lr_X_Voltage >= DINT_TO_REAL(adi_X_MeasurePoint_Voltage[ii])) AND (lr_X_Voltage <= DINT_TO_REAL(adi_X_MeasurePoint_Voltage[ii + 1])) THEN
			IF ((adi_X_MeasurePoint_Voltage[ii+1] - adi_X_MeasurePoint_Voltage[ii]) <> 0.0) THEN
				lr_M_gradient:=(DINT_TO_REAL(adi_X_FixedValue[ii+1]) - DINT_TO_REAL(adi_X_FixedValue[ii])) / (DINT_TO_REAL(adi_X_MeasurePoint_Voltage[ii+1]) - DINT_TO_REAL(adi_X_MeasurePoint_Voltage[ii]));	(* Berechnung der Steigung m *)
			END_IF;
			lr_B_AxisIntercept:=DINT_TO_REAL(adi_X_FixedValue[ii]) - (lr_M_gradient * DINT_TO_REAL(adi_X_MeasurePoint_Voltage[ii]));	(* berechnung des Y-Achsenabschnittes *)
			EXIT;
		END_IF;
	END_FOR;
	IF (ii <= 9) THEN
		IF (lr_M_gradient <> 0.0) THEN
			lrScaledValuePercent:=(lr_M_gradient * lr_X_Voltage) + lr_B_AxisIntercept;	(* Lineare Funktion-->ausrechnen des linearisierten Kraft *)
		END_IF;
	ELSE
		IF (lr_X_Voltage > adi_X_MeasurePoint_Voltage[10]) THEN
			lrScaledValuePercent:=DINT_TO_LREAL(adi_X_FixedValue[10]);
		ELSE
			lrScaledValuePercent:=DINT_TO_REAL(adi_X_FixedValue[0]);
		END_IF;
	END_IF;
ELSE
	lrScaledValuePercent:=DINT_TO_REAL(adi_X_FixedValue[0]);
END_IF;
IF (lrScaledValuePercent < DINT_TO_REAL(adi_X_FixedValue[0])) THEN
	lrScaledValuePercent:=DINT_TO_REAL(adi_X_FixedValue[0]);
END_IF;
IF (lrScaledValuePercent > DINT_TO_REAL(adi_X_FixedValue[10])) THEN
	lrScaledValuePercent:=DINT_TO_REAL(adi_X_FixedValue[10]);
END_IF;
lrScaledValuePercent:=DINT_TO_LREAL(LREAL_TO_DINT(lrScaledValuePercent));
lrValuePercent:=REAL_TO_BYTE((100.0/32768.0) * lr_X_Voltage);	(* Nicht linearisierter Wert-->0% bis 100% *)
IF (lrValuePercent < DINT_TO_REAL(adi_X_FixedValue[0])) THEN
	lrValuePercent:=DINT_TO_REAL(adi_X_FixedValue[0]);
END_IF;
IF (lrValuePercent > DINT_TO_REAL(adi_X_FixedValue[10])) THEN
	lrValuePercent:=DINT_TO_REAL(adi_X_FixedValue[10]);
END_IF;
END_FUNCTION_BLOCK

(* POU PRG_LAYER5_VISU/FB_VISU/Function/FB_TeachPosToHMI, ST *)
FUNCTION_BLOCK FB_TeachPosToHMI
(*Bearb-Station: Zuweisung der Teach-Werte zur HMI-Struct*)
VAR_INPUT
	iAxisNr				:INT;
	iSelectPos			:INT;
	rSetPos				:REAL;(*Input from HMI-Var: SetPos*)

	TeachPosWork		: ST_EXCHG_PARAM_STANDARDPROCESS;
END_VAR
VAR_OUTPUT
	rPosition				:REAL;
END_VAR
VAR
END_VAR
IF NOT(T_NovRam.T_Parameter.T_StationWork[1].T_StProcess.xConfigActive) THEN
		CASE iAxisNr OF
		(* Z Axis *)
		1:	CASE iSelectPos OF
			(* < Fahre zu man. Pos. > *)
			0:	rPosition:=rSetPos;
			(* < Z LadePos > *)
			1:	rPosition:=TeachPosWork.rPositionLoad;
			(* < Z Bearb StartPos > *)
			2:	rPosition:=TeachPosWork.rPositionStartProc;
			(* < Z ZentrierPos > *)
			3:	rPosition:=TeachPosWork.rCentringPosZ1Axis;
			(* < Z Bearb EndPos > *)
			4:	rPosition:=TeachPosWork.rPositionEndProc;
			(* < Z WzWechsel Pos > *)
			5:	rPosition:=TeachPosWork.rPositionToolChange;
			(* < Z Mech EndPos > *)
			6:	rPosition:=TeachPosWork.rPositionEndMech;
			(* < Z Bearb EndPos berechn. > *)
			7:	rPosition:=garPositionEndProcCalc[1];
			(* < Z Bearb EndPos Max > *)
			8:	rPosition:=TeachPosWork.rPositionEndProcMaxInc;
			(* < Z ZentrierPos berechn. > *)
			9:	rPosition:=garCentringEndProcCalc[1];
			(* < Z WzZylinder Pos > *)
			10:	rPosition:=TeachPosWork.rZPositionCylindricalArea;
			END_CASE;
		END_CASE;
ELSE
		CASE iAxisNr OF
		(* Z Axis *)
		1:	CASE iSelectPos OF
			(* < Fahre zu man. Pos. > *)
			0:	rPosition:=rSetPos;
			(* < Z LadePos > *)
			1:	rPosition:=grZ_LoadPos;
			(* < Z Bearb StartPos > *)
			2:	rPosition:=grZ_WorkStartPos;
			(* < Z ZentrierPos > *)
			3:	rPosition:=TeachPosWork.rCentringPosZ1Axis;
			(* < Z Bearb EndPos > *)
			4:	rPosition:=garPositionEndProcCalc[1];
			(* < Z WzWechsel Pos > *)
			5:	rPosition:=TeachPosWork.rPositionToolChange;
			(* < Z Mech EndPos > *)
			6:	rPosition:=TeachPosWork.rPositionEndMech;
			(* < Z Bearb EndPos berechn. > *)
			7:	rPosition:=garPositionEndProcCalc[1];
			(* < Z Bearb EndPos Max > *)
			8:	rPosition:=TeachPosWork.rPositionEndProcMaxInc;
			(* < Z ZentrierPos berechn. > *)
			9:	rPosition:=garCentringEndProcCalc[1];
			(* < Z WzZylinder Pos > *)
			10:	rPosition:=TeachPosWork.rZPositionCylindricalArea;
			END_CASE;
		END_CASE;
END_IF;
END_FUNCTION_BLOCK

(* POU PRG_LAYER5_VISU/FB_VISU/Function/FB_GetStationFunctionNr, ST *)
FUNCTION_BLOCK FB_GetStationFunctionNr
VAR_INPUT
	iVisuFunctionNr:INT;
END_VAR
VAR_OUTPUT
	iWorkStation_FunctionNr:INT;
END_VAR
VAR
END_VAR
iWorkStation_FunctionNr:=0;
CASE iVisuFunctionNr OF
(* < Grundstellungsfahrt BearbStation > *)
1:	iWorkStation_FunctionNr:=2;
(* < S Axis EIN > *)
2:	iWorkStation_FunctionNr:=3;
(* < Wz Einfädeln > *)
3:	iWorkStation_FunctionNr:=4;
(* < Wstk Zentrieren > *)
4:	iWorkStation_FunctionNr:=11;
(* < Bearbeitungsprozess > *)
5:	iWorkStation_FunctionNr:=5;
(* < S Axis AUS > *)
6:	iWorkStation_FunctionNr:=6;
END_CASE;
END_FUNCTION_BLOCK

(* POU PRG_LAYER5_VISU/FB_VISU/Function/iFct_GetLeftButtonNumber, ST *)
FUNCTION iFct_GetLeftButtonNumber : INT
VAR_INPUT
	dwActualPage:DWORD;
END_VAR
VAR
	iTmpLeftButtonNumber:INT;
END_VAR
iFct_GetLeftButtonNumber:=iTmpLeftButtonNumber:=0;
IF ((dwActualPage >= 10) AND (dwActualPage <= 99)) THEN
	iTmpLeftButtonNumber:=0;	(* No Button active *)
	IF (dwActualPage = 70) THEN
		iTmpLeftButtonNumber:=iTmpLeftButtonNumber + 16;	(* Parameter Button active *)
	END_IF;
END_IF;
IF ((dwActualPage >= 100) AND (dwActualPage <= 199)) THEN
	iTmpLeftButtonNumber:=1;	(* Button 1 active *)
	IF (dwActualPage = 170) THEN
		iTmpLeftButtonNumber:=iTmpLeftButtonNumber + 16;	(* Button 1 and Parameter Button active *)
	END_IF;
END_IF;
IF ((dwActualPage >= 200) AND (dwActualPage <= 299)) THEN
	iTmpLeftButtonNumber:=2;	(* Button 2 active *)
	IF (dwActualPage = 270) THEN
		iTmpLeftButtonNumber:=iTmpLeftButtonNumber + 16;	(* Button 2 and Parameter Button active *)
	END_IF;
END_IF;
IF ((dwActualPage >= 300) AND (dwActualPage <= 399)) THEN
	iTmpLeftButtonNumber:=4;	(* Button 3 active *)
	IF (dwActualPage = 370) THEN
		iTmpLeftButtonNumber:=iTmpLeftButtonNumber + 16;	(* Button 3 and Parameter Button active *)
	END_IF;
END_IF;
IF ((dwActualPage >= 400) AND (dwActualPage <= 499)) THEN
	iTmpLeftButtonNumber:=8;	(* Button 1 active *)
	IF (dwActualPage = 470) THEN
		iTmpLeftButtonNumber:=iTmpLeftButtonNumber + 16;	(* Button 4 and Parameter Button active *)
	END_IF;
END_IF;
iFct_GetLeftButtonNumber:=iTmpLeftButtonNumber;
END_FUNCTION

(* POU PRG_LAYER5_VISU/FB_VISU/Function/xFct_GetParameterPageActive, ST *)
FUNCTION xFct_GetParameterPageActive : BOOL
VAR_INPUT
	dwActualPage:DWORD;
END_VAR
VAR
END_VAR
xFct_GetParameterPageActive:=FALSE;
IF (dwActualPage = 70) OR (dwActualPage = 170) OR (dwActualPage = 270) OR (dwActualPage = 370) OR (dwActualPage = 470) THEN
	xFct_GetParameterPageActive:=TRUE;
END_IF;
END_FUNCTION

(* POU PRG_LAYER5_VISU/FB_VISU/Function/wFct_GetTaskNumber, ST *)
FUNCTION wFct_GetTaskNumber : WORD
VAR_INPUT
	dwActualPage:DWORD;
END_VAR
VAR
	wTmpTaskNumber: WORD;
END_VAR
wFct_GetTaskNumber:=wTmpTaskNumber:=1;
IF ((dwActualPage >= 10) AND (dwActualPage <= 19)) OR ((dwActualPage >= 110) AND (dwActualPage <= 119)) OR
     ((dwActualPage >= 210) AND (dwActualPage <= 219)) OR ((dwActualPage >= 310) AND (dwActualPage <= 319)) OR ((dwActualPage >= 410) AND (dwActualPage <= 419)) THEN
	wTmpTaskNumber:=1;	(* Task 1 *)
END_IF;
IF ((dwActualPage >= 20) AND (dwActualPage <= 29)) OR ((dwActualPage >= 120) AND (dwActualPage <= 129)) OR
     ((dwActualPage >= 220) AND (dwActualPage <= 229)) OR ((dwActualPage >= 320) AND (dwActualPage <= 329)) OR ((dwActualPage >= 420) AND (dwActualPage <= 429)) THEN
	wTmpTaskNumber:=2;	(* Task 2 *)
END_IF;
IF ((dwActualPage >= 30) AND (dwActualPage <= 39)) OR ((dwActualPage >= 130) AND (dwActualPage <= 139)) OR
     ((dwActualPage >= 230) AND (dwActualPage <= 239)) OR ((dwActualPage >= 330) AND (dwActualPage <= 339)) OR ((dwActualPage >= 430) AND (dwActualPage <= 439)) THEN
	wTmpTaskNumber:=4;	(* Task 3 *)
END_IF;
IF ((dwActualPage >= 40) AND (dwActualPage <= 49)) OR ((dwActualPage >= 140) AND (dwActualPage <= 149)) OR
     ((dwActualPage >= 240) AND (dwActualPage <= 249)) OR ((dwActualPage >= 340) AND (dwActualPage <= 349)) OR ((dwActualPage >= 440) AND (dwActualPage <= 449)) THEN
	wTmpTaskNumber:=8;	(* Task 4 *)
END_IF;
IF ((dwActualPage >= 50) AND (dwActualPage <= 59)) OR ((dwActualPage >= 150) AND (dwActualPage <= 159)) OR
     ((dwActualPage >= 250) AND (dwActualPage <= 259)) OR ((dwActualPage >= 350) AND (dwActualPage <= 359)) OR ((dwActualPage >= 450) AND (dwActualPage <= 459)) THEN
	wTmpTaskNumber:=16;	(* Task 5 *)
END_IF;
IF ((dwActualPage >= 60) AND (dwActualPage <= 69)) OR ((dwActualPage >= 160) AND (dwActualPage <= 169)) OR
     ((dwActualPage >= 260) AND (dwActualPage <= 269)) OR ((dwActualPage >= 360) AND (dwActualPage <= 369)) OR ((dwActualPage >= 460) AND (dwActualPage <= 469)) THEN
	wTmpTaskNumber:=32;	(* Task 6 *)
END_IF;
wFct_GetTaskNumber:=wTmpTaskNumber;
END_FUNCTION

(* POU PRG_LAYER5_VISU/FB_VISU/Function/xFct_SetActualPageTask, ST *)
FUNCTION xFct_SetActualPageTask : BOOL
VAR_INPUT
	dwActualPage:DWORD;
	iTaskBarNumber:INT;
END_VAR
VAR_IN_OUT
	dwSaveActualPageTask:ARRAY [0..4,1..6] OF DWORD;
END_VAR
VAR
END_VAR
IF ((dwActualPage >= 10) AND (dwActualPage <= 69)) THEN
	dwSaveActualPageTask[0,iTaskBarNumber]:=dwActualPage;
END_IF;
IF ((dwActualPage >= 110) AND (dwActualPage <= 169)) THEN
	dwSaveActualPageTask[1,iTaskBarNumber]:=dwActualPage;
END_IF;
IF ((dwActualPage >= 210) AND (dwActualPage <= 269)) THEN
	dwSaveActualPageTask[2,iTaskBarNumber]:=dwActualPage;
END_IF;
IF ((dwActualPage >= 310) AND (dwActualPage <= 369)) THEN
	dwSaveActualPageTask[3,iTaskBarNumber]:=dwActualPage;
END_IF;
IF ((dwActualPage >= 410) AND (dwActualPage <= 469)) THEN
	dwSaveActualPageTask[4,iTaskBarNumber]:=dwActualPage;
END_IF;
END_FUNCTION

(* POU PRG_LAYER5_VISU/FB_VISU/Function/xFct_CheckSingleButtonActivation, ST *)
FUNCTION xFct_CheckSingleButtonActivation : BOOL
VAR_INPUT
	wInputButton:WORD;
END_VAR
VAR
	wTmp:WORD;
	ii: INT;
	iCountNumberButtonActivation: INT;
END_VAR
(* Return TRUE if only one button is pressed *)
xFct_CheckSingleButtonActivation:=FALSE;
wTmp:=wInputButton;
iCountNumberButtonActivation:=0;
FOR  ii:=1 TO 16 DO	(* Only for datatype WORD-->16Bit *)
	IF (wTmp AND 16#1) = 16#1 THEN
		iCountNumberButtonActivation:=iCountNumberButtonActivation + 1;
	END_IF;
	wTmp:=ROR(wTmp,1);	(* Shift 1 Bit to right *)
END_FOR;
IF (iCountNumberButtonActivation = 1) THEN
	xFct_CheckSingleButtonActivation:=TRUE;
END_IF;
END_FUNCTION

(* POU PRG_LAYER5_VISU/FB_VISU/Function/xFct_GetJogMode, ST *)
FUNCTION xFct_GetJogMode : BOOL
VAR_INPUT
	iFunction:INT;		(* Übergabe der Visualisierungsfunktionsnummer *)
END_VAR
VAR
	xJogModeActive: BOOL;
END_VAR
xJogModeActive:=FALSE;
IF (iFunction = 216) THEN	(* Achse Jog/Ink Bewegung -/- - *)
	xJogModeActive:=TRUE;
ELSIF (iFunction = 217) THEN	(* Achse Jog/Ink Bewegung +/++ *)
	xJogModeActive:=TRUE;
END_IF;
xFct_GetJogMode:=xJogModeActive;
END_FUNCTION

(* POU PRG_LAYER5_VISU/FB_VISU/Function/xFct_GetNormalOperateActive, ST *)
FUNCTION xFct_GetNormalOperateActive : BOOL
VAR_INPUT
	dwActualPage:DWORD;
END_VAR
VAR
END_VAR
xFct_GetNormalOperateActive:=FALSE;
IF (dwActualPage >= 10) AND (dwActualPage <= 99) THEN
	xFct_GetNormalOperateActive:=TRUE;
END_IF;
END_FUNCTION

(* POU PRG_LAYER5_VISU/FB_VISU/Function/xFct_GetSetupOperateActive, ST *)
FUNCTION xFct_GetSetupOperateActive : BOOL
VAR_INPUT
	dwActualPage:DWORD;
END_VAR
VAR
END_VAR
xFct_GetSetupOperateActive:=FALSE;
IF (dwActualPage >= 110) AND (dwActualPage <= 499) THEN
	xFct_GetSetupOperateActive:=TRUE;
END_IF;
END_FUNCTION

(* POU PRG_LAYER5_VISU/FB_VISU/Function/xFct_GetSetupMode, ST *)
FUNCTION xFct_GetSetupMode : BOOL
VAR_INPUT
	dwActualPage:DWORD;
	iSetupModeRequest:INT;
END_VAR
VAR
END_VAR
xFct_GetSetupMode:=FALSE;
IF (iSetupModeRequest = 1) THEN
	IF (dwActualPage >= 110) AND (dwActualPage <= 199) THEN
		xFct_GetSetupMode:=TRUE;
	END_IF;
END_IF;
IF (iSetupModeRequest = 2) THEN
	IF (dwActualPage >= 210) AND (dwActualPage <= 299) THEN
		xFct_GetSetupMode:=TRUE;
	END_IF;
END_IF;
IF (iSetupModeRequest = 3) THEN
	IF (dwActualPage >= 310) AND (dwActualPage <= 399) THEN
		xFct_GetSetupMode:=TRUE;
	END_IF;
END_IF;
IF (iSetupModeRequest = 4) THEN
	IF (dwActualPage >= 410) AND (dwActualPage <= 499) THEN
		xFct_GetSetupMode:=TRUE;
	END_IF;
END_IF;
END_FUNCTION

(* POU PRG_LAYER5_VISU/FB_VISU/Function/bFct_GetLedState, ST *)
FUNCTION bFct_GetLedState : BYTE
VAR_INPUT
	iLampNumber:INT;
END_VAR
VAR
END_VAR
IF (iLampNumber = 1) THEN
	bFct_GetLedState:=1;
ELSIF (iLampNumber = 2) THEN
	bFct_GetLedState:=2;
ELSIF (iLampNumber = 3) THEN
	bFct_GetLedState:=3;
ELSIF (iLampNumber = 4) THEN
	bFct_GetLedState:=4;
ELSIF (iLampNumber = 5) THEN
	bFct_GetLedState:=5;
ELSIF (iLampNumber = 13) THEN
	bFct_GetLedState:=1;
ELSIF (iLampNumber = 14) THEN
	bFct_GetLedState:=3;
ELSIF (iLampNumber = 15) THEN
	bFct_GetLedState:=2;
ELSIF (iLampNumber = 16) THEN
	bFct_GetLedState:=1;
END_IF;
END_FUNCTION

(* POU PRG_LAYER5_VISU/FB_VISU/Function/sFct_GetLampOrderNumberEngl, ST *)
FUNCTION sFct_GetLampOrderNumberEngl : STRING(90)
VAR_INPUT
	xLampdefect:BOOL;
	iLampNumber:INT;
END_VAR
VAR
END_VAR
sFct_GetLampOrderNumberEngl:='';
IF xLampdefect THEN
	IF (iLampNumber = 1) THEN
		sFct_GetLampOrderNumberEngl:='Microcut order no.: 986.03.03.001:   LED-Element 24VDC green(Start Button)';
	ELSIF (iLampNumber = 2) THEN
		sFct_GetLampOrderNumberEngl:='Microcut order no.: 986.03.03.003:   LED-Element 24VDC red(Stop Button)';
	ELSIF (iLampNumber = 3) THEN
		sFct_GetLampOrderNumberEngl:='Microcut order no.: 986.03.03.004:   LED-Element 24VDC white(Axislocking Button)';
	ELSIF (iLampNumber = 4) THEN
		sFct_GetLampOrderNumberEngl:='Microcut order no.: 986.03.03.002:   LED-Element 24VDC blue(Enabling Button)';
	ELSIF (iLampNumber = 5) THEN
		sFct_GetLampOrderNumberEngl:='Microcut order no.: 986.03.03.004:   LED-Element 24VDC yellow(SetupMode Lamp)';
	ELSIF (iLampNumber = 13) THEN
		sFct_GetLampOrderNumberEngl:='Microcut order no.: 986.06.04.025:   Control lamp (green)';
	ELSIF (iLampNumber = 14) THEN
		sFct_GetLampOrderNumberEngl:='Microcut order no.: 986.06.04.025:   Control lamp (yellow)';
	ELSIF (iLampNumber = 15) THEN
		sFct_GetLampOrderNumberEngl:='Microcut order no.: 986.06.04.025:   Control lamp (red)';
	ELSIF (iLampNumber = 16) THEN
		sFct_GetLampOrderNumberEngl:='Microcut order no.: 986.06.04.026:   Indoor Lamp';
	END_IF;
ELSE
	IF (iLampNumber = 1) THEN
		sFct_GetLampOrderNumberEngl:='LED-Element 24VDC green(Start Button)';
	ELSIF (iLampNumber = 2) THEN
		sFct_GetLampOrderNumberEngl:='LED-Element 24VDC red(Stop Button)';
	ELSIF (iLampNumber = 3) THEN
		sFct_GetLampOrderNumberEngl:='LED-Element 24VDC white(Axislocking Button)';
	ELSIF (iLampNumber = 4) THEN
		sFct_GetLampOrderNumberEngl:='LED-Element 24VDC blue(Enabling Button)';
	ELSIF (iLampNumber = 5) THEN
		sFct_GetLampOrderNumberEngl:='LED-Element 24VDC yellow(SetupMode Lamp)';
	ELSIF (iLampNumber = 13) THEN
		sFct_GetLampOrderNumberEngl:='Control lamp (green)';
	ELSIF (iLampNumber = 14) THEN
		sFct_GetLampOrderNumberEngl:='Control lamp (yellow)';
	ELSIF (iLampNumber = 15) THEN
		sFct_GetLampOrderNumberEngl:='Control lamp (red)';
	ELSIF (iLampNumber = 16) THEN
		sFct_GetLampOrderNumberEngl:='Indoor Lamp';
	END_IF;
END_IF;
END_FUNCTION

(* POU PRG_LAYER5_VISU/FB_VISU/Function/sFct_GetLampOrderNumberGer, ST *)
FUNCTION sFct_GetLampOrderNumberGer : STRING(90)
VAR_INPUT
	xLampdefect:BOOL;
	iLampNumber:INT;
END_VAR
VAR
END_VAR
sFct_GetLampOrderNumberGer:='';
IF xLampdefect THEN
	IF (iLampNumber = 1) THEN
		sFct_GetLampOrderNumberGer:='Microcut BestellNr.: 986.03.03.001:   LED-Element 24VDC grün(Start Taste)';
	ELSIF (iLampNumber = 2) THEN
		sFct_GetLampOrderNumberGer:='Microcut BestellNr.: 986.03.03.003:   LED-Element 24VDC rot(Stopp Taste)';
	ELSIF (iLampNumber = 3) THEN
		sFct_GetLampOrderNumberGer:='Microcut BestellNr.: 986.03.03.004:   LED-Element 24VDC weiss(Achsensperr Taste)';
	ELSIF (iLampNumber = 4) THEN
		sFct_GetLampOrderNumberGer:='Microcut BestellNr.: 986.03.03.002:   LED-Element 24VDC blau(Freigabe Taste)';
	ELSIF (iLampNumber = 5) THEN
		sFct_GetLampOrderNumberGer:='Microcut BestellNr.: 986.03.03.004:   LED-Element 24VDC gelb(Einrichtlampe)';
	ELSIF (iLampNumber = 13) THEN
		sFct_GetLampOrderNumberGer:='Microcut BestellNr.: 986.06.04.025:   Kontrolllampe (grün)';
	ELSIF (iLampNumber = 14) THEN
		sFct_GetLampOrderNumberGer:='Microcut BestellNr.: 986.06.04.025:   Kontrolllampe (gelb)';
	ELSIF (iLampNumber = 15) THEN
		sFct_GetLampOrderNumberGer:='Microcut BestellNr.: 986.06.04.025:   Kontrolllampe (rot)';
	ELSIF (iLampNumber = 16) THEN
		sFct_GetLampOrderNumberGer:='Microcut BestellNr.: 986.06.04.026:   Maschinenlampe';
	END_IF;
ELSE
	IF (iLampNumber = 1) THEN
		sFct_GetLampOrderNumberGer:='LED-Element 24VDC grün(Start Taste)';
	ELSIF (iLampNumber = 2) THEN
		sFct_GetLampOrderNumberGer:='LED-Element 24VDC rot(Stopp Taste)';
	ELSIF (iLampNumber = 3) THEN
		sFct_GetLampOrderNumberGer:='LED-Element 24VDC weiss(Achsensperr Taste)';
	ELSIF (iLampNumber = 4) THEN
		sFct_GetLampOrderNumberGer:='LED-Element 24VDC blau(Freigabe Taste)';
	ELSIF (iLampNumber = 5) THEN
		sFct_GetLampOrderNumberGer:='LED-Element 24VDC gelb(Einrichtlampe)';
	ELSIF (iLampNumber = 13) THEN
		sFct_GetLampOrderNumberGer:='Kontrolllampe (grün)';
	ELSIF (iLampNumber = 14) THEN
		sFct_GetLampOrderNumberGer:='Kontrolllampe (gelb)';
	ELSIF (iLampNumber = 15) THEN
		sFct_GetLampOrderNumberGer:='Kontrolllampe (rot)';
	ELSIF (iLampNumber = 16) THEN
		sFct_GetLampOrderNumberGer:='Maschinenlampe';
	END_IF;
END_IF;
END_FUNCTION

(* POU GENERAL/PROFILE/iFctExistProfileName, ST *)
FUNCTION iFctExistProfileName : INT
VAR_INPUT
	sProfileName:STRING(30);
	ptrProfileList:POINTER TO ARRAY[1..4,1..csiMaxProfile] OF ST_PROFILE_ID;
END_VAR
VAR
	i:INT;
	sTmp:STRING;
	sTmp2:STRING;
END_VAR
(* Init. function *)
	iFctExistProfileName:=0;
	sTmp:=sFctUpLowCase(	xLowConvert:=TRUE,
							sInString:=sProfileName);

(* Search if name already exists *)
	FOR i:=1 TO csiMaxProfile DO
		sTmp2:=	sFctUpLowCase(	xLowConvert:=TRUE,
								sInString:=ptrProfileList^[gciStationSt1,i].sName);
		IF sTmp = sTmp2 AND sTmp2 <> '' THEN iFctExistProfileName:=i; RETURN; END_IF
	END_FOR
END_FUNCTION

(* POU GENERAL/sFctUpLowCase, ST *)
FUNCTION sFctUpLowCase : STRING
VAR_INPUT
	xLowConvert:BOOL;
	sInString:STRING;
END_VAR
VAR
(* variable *)
	sListUpCase:STRING:='ABCDEFGHIJKLMNOPQRSTUVWXYZ';
	sListLowCase:STRING:='abcdefghijklmnopqrstuvwxyz';
	i:INT;
(* Tmp *)
	sTmp:STRING;
	iTmp:INT;
END_VAR
(* Init. *)
	sFctUpLowCase:='';

(*Test string size*)
	IF LEN(sInString) < 1 OR LEN(sInString) > 255 THEN RETURN; END_IF

	IF xLowConvert THEN
	(* Conversion to low case *)
		FOR i:= 1 TO LEN(sInString) DO
			sTmp:=MID(sInString,1,i);
			iTmp:=FIND(sListUpCase,sTmp);
			IF iTmp > 0 THEN sFctUpLowCase:=CONCAT(sFctUpLowCase,MID(sListLowCase,1,iTmp));
				ELSE sFctUpLowCase:=CONCAT(sFctUpLowCase,sTmp); END_IF
		END_FOR
	(* Conversion to up case *)
	ELSE
		FOR i:= 1 TO LEN(sInString) DO
			sTmp:=MID(sInString,1,i);
			iTmp:=FIND(sListLowCase,sTmp);
			IF iTmp > 0 THEN sFctUpLowCase:=CONCAT(sFctUpLowCase,MID(sListUpCase,1,iTmp));
				ELSE sFctUpLowCase:=CONCAT(sFctUpLowCase,sTmp); END_IF
		END_FOR
	END_IF
END_FUNCTION

(* POU GENERAL/FB_CTRLEBUTTON, ST *)
FUNCTION_BLOCK FB_CTRLEBUTTON
VAR_INPUT
	xReadyFB:BOOL;
	xHWStart:BOOL;
	xHWStop:BOOL;
	dwActualPage:DWORD;
	T_VisuQVis:ST_QVIS;
	T_ExchgParam:ST_QVIS_EXCHG_PARAM;
	xSecurityKey:BOOL;		(* state of the keyswitch-->TRUE=EinrichtBetrieb *)
	iSetupMode:INT;			(* Turn switch --> 1=EinrichtBetriebA, 2=EinrichtBetriebB *)
	xNormalOperate_EnergyON:BOOL;
	xSetupOperateA_EnergyON:BOOL;
	xSetupOperateB_EnergyON:BOOL;
	xSetupOperateC_EnergyON:BOOL;
END_VAR
VAR_OUTPUT
END_VAR
VAR_IN_OUT
	T_StartButton: ST_BUTTON;
	T_StopButton:ST_BUTTON;
END_VAR
VAR
(* Variable *)
	iIndexActivPage:INT;
(* FB Mask *)
	xMaskPageBtStart:BOOL;
	xMaskPageBtStop:BOOL;
(* Trigger *)
	RisingEdgeSignalStartButton:R_TRIG;
	RisingEdgeSignalStopButton:R_TRIG;
(* Tmp variable *)
	xTmp:BOOL;
	xNotCheckState: BOOL;
	xProcessReady: BOOL;
	xVisuActionReady: BOOL;
	xNotCheckStateStop: BOOL;
	xProcessActive: BOOL;
	xStationReady_SetupMode1: BOOL;
	xStationReady_SetupMode2: BOOL;
	xStationReady_NormalMode: BOOL;
	xStationSecurityStateON: BOOL;
END_VAR
(* exit FB if machine is not start up and ready *)
	IF NOT(xReadyFB) THEN RETURN;	END_IF;

(* Index Activ Page *)
	iIndexActivPage:=T_VisuQVis.T_PageIndex[dwActualPage].iIndexConfigPage;
	xMaskPageBtStart:=FALSE;
	xMaskPageBtStop:=FALSE;


	xProcessReady:=	NOT(TProcess.T_Ctrle.xExecute) AND TProcess.T_Ctrle.xDone AND NOT(T_VisuQVis.T_CtrleProcess.xExecute) AND T_VisuQVis.T_CtrleProcess.xDone;
	xProcessActive:=	(NOT(TProcess.T_Ctrle.xExecute) AND NOT(TProcess.T_Ctrle.xDone)) OR
						(NOT(T_VisuQVis.T_CtrleProcess.xExecute) AND NOT(T_VisuQVis.T_CtrleProcess.xDone) AND NOT(T_VisuQVis.T_CtrleProcess.xErr));

	xStationSecurityStateON:=	TStation_Work_St1.TControl.xSecurityCircuitOn;


	xStationReady_SetupMode1:=	(TStation_Work_St1.TControl.xDone AND TStation_Work_St1.TControl.xRdy AND NOT(TStation_Work_St1.TControl.xError)) AND
									xSetupOperateA_EnergyON;

	xStationReady_SetupMode2:=	(TStation_Work_St1.TControl.xDone AND TStation_Work_St1.TControl.xRdy AND NOT(TStation_Work_St1.TControl.xError)) AND
									xSetupOperateB_EnergyON;

	xStationReady_NormalMode:=	xStationReady_SetupMode1 AND xStationReady_SetupMode2 AND xNormalOperate_EnergyON;

	xVisuActionReady:=NOT(T_VisuQVis.T_CtrleAction.xExecute) AND T_VisuQVis.T_CtrleAction.xDone;

	IF NOT(xSecurityKey) THEN
		xNotCheckState:=		NOT(xNormalOperate_EnergyON) OR (T_ExchgParam.T_Visu.bMachineState = 4) OR
								(T_ExchgParam.T_SafetyCtrl.bStateMessageError <> 0) OR (T_ExchgParam.T_SafetyCtrl.bStateMessageInfo <> 0) OR
								(T_ExchgParam.T_SafetyCtrl.bStateMessageWarning <> 0) OR NOT(xProcessReady) OR NOT(xVisuActionReady) OR NOT(xStationReady_NormalMode);
		xNotCheckStateStop:=	NOT(xNormalOperate_EnergyON) OR (T_ExchgParam.T_Visu.bMachineState = 4) OR
								(T_ExchgParam.T_SafetyCtrl.bStateMessageError <> 0) OR (T_ExchgParam.T_SafetyCtrl.bStateMessageInfo <> 0) OR
								(T_ExchgParam.T_SafetyCtrl.bStateMessageWarning <> 0);
	ELSE
		IF (iSetupMode = 1) THEN
			xNotCheckState:=	NOT(xSetupOperateA_EnergyON) OR (T_ExchgParam.T_Visu.bMachineState = 4) OR NOT(xProcessReady) OR NOT(xVisuActionReady) OR NOT(xStationReady_SetupMode1);
			xNotCheckStateStop:=NOT(xSetupOperateA_EnergyON) OR (T_ExchgParam.T_Visu.bMachineState = 4);
		ELSIF (iSetupMode = 2) THEN
			xNotCheckState:=	NOT(xSetupOperateB_EnergyON) OR (T_ExchgParam.T_Visu.bMachineState = 4) OR NOT(xVisuActionReady) OR NOT(xStationReady_SetupMode2);
			xNotCheckStateStop:=NOT(xSetupOperateB_EnergyON) OR (T_ExchgParam.T_Visu.bMachineState = 4);
		ELSE
			xNotCheckState:=TRUE;
		END_IF;
	END_IF;
(* Start Button *)
	IF NOT(xNotCheckState) OR T_CtrleBtStartStop.xForceSetStartButton THEN
		CASE dwActualPage OF
		gT_PageNumber.iAutoMode_Process, gT_PageNumber.iAutoMode_ProcessValue1, gT_PageNumber.iAutoMode_ProcessValue2, gT_PageNumber.iAutoMode_PartQuality:		(* Automat Prozess *)
			xMaskPageBtStart:=TRUE;
			IF T_CtrleBtStartStop.xForceSetStartButton THEN
				xMaskPageBtStart:=TRUE;
			END_IF;
		gT_PageNumber.iAutoMode_Referencing:	(* Maschinenreferenzierung Prozess *)
			xMaskPageBtStart:=TRUE;
		gT_PageNumber.iHandMode_Process,gT_PageNumber.iHandMode_WorkParameter,gT_PageNumber.iHandMode_RegulatorPara,gT_PageNumber.iHandMode_OnlineChange,gT_PageNumber.iHandMode_ConfigPosition:		(* HandBetrieb Prozess *)
			xMaskPageBtStart:=TRUE;
			IF T_CtrleBtStartStop.xForceSetStartButton THEN
				xMaskPageBtStart:=TRUE;
			END_IF;
		gT_PageNumber.iWorkStation_Axis1:		(* TeachIN für Absolut Bewegung oder Geschwindigkeitsbewegung *)
			IF (T_ExchgParam.T_StationCommon.wState AND 16#6) = 16#0 THEN
				(* Station darf nicht Aktiv sein und kein Fehler darf vorhanden sein *)
				CASE T_ExchgParam.T_TeachIn.iSetup_AxisSel OF
				gciAxisZ_St1:
					IF (T_ExchgParam.T_TeachIn.arAxis[gciAxisZ_St1].bActState AND 16#F) = 16#3 THEN
						xMaskPageBtStart:=TRUE;	(* Achse muss Referenziert sein, Achsenstrom muss eingeschaltet sein, kein Fehler und Achse darf sich nicht bewegen *)
					END_IF;
				gciAxisS_St1,3:
					IF (T_ExchgParam.T_TeachIn.arAxis[gciAxisS_St1].bActState AND 16#F) = 16#1 THEN
						xMaskPageBtStart:=TRUE;	(* Achse muss Referenziert sein, Achsenstrom muss eingeschaltet sein, kein Fehler und Achse darf sich nicht bewegen *)
					END_IF;
				END_CASE;
			END_IF;
		gT_PageNumber.iWorkStation_Function1:		(* Ausführen von Stationsfunktionen der Bearbeitungsstation MicroHead und EntgratStation *)
			IF ((T_ExchgParam.T_StationCommon.wState AND 16#6) = 16#0) THEN
				(* Stationen Bearb, Lade/Entlade und Teller dürfen nicht Aktiv sein und kein Fehler darf vorhanden sein *)
				xMaskPageBtStart:=TRUE;
			END_IF;
			IF T_CtrleBtStartStop.xForceSetStartButton THEN
				xMaskPageBtStart:=TRUE;
			END_IF;
		gT_PageNumber.iWorkStation_Setup1:		(* Ausführen der Stationsfunktion für das Kalibrieren des ToolDefelction und ToolTorque *)
			IF ((T_ExchgParam.T_StationCommon.wState AND 16#6) = 16#0) THEN
				(* Station Bearb darf nicht Aktiv sein und kein Fehler darf vorhanden sein *)
				xMaskPageBtStart:=TRUE;
			END_IF;
		gT_PageNumber.iWorkStation_Setup2:		(* Ausführen der Stationsfunktion für das Kalibrieren des ToolDefelction und ToolTorque *)
			IF ((T_ExchgParam.T_StationCommon.wState AND 16#6) = 16#0) THEN
				(* Station Bearb darf nicht Aktiv sein und kein Fehler darf vorhanden sein *)
				xMaskPageBtStart:=TRUE;
			END_IF;
		gT_PageNumber.iWorkStation_Setup3:			(* Ausführen von Stationsfunktionen für das Einrichten der Z Achse für die erst einrichtung *)
			IF (T_ExchgParam.T_StationCommon.iZAxisFirstSetup_StepNr = 1) THEN
				IF (T_ExchgParam.T_StationCommon.wState AND 16#6) = 16#0 THEN
					(* Arbeitsstation darf nicht Aktiv sein und kein Fehler darf vorhanden sein *)
					xMaskPageBtStart:=TRUE;
				END_IF;
			END_IF;
			IF T_CtrleBtStartStop.xForceSetStartButton THEN
				xMaskPageBtStart:=TRUE;
			END_IF;
		END_CASE;

		IF (T_ExchgParam.T_Visu.T_Message.iState = 401) THEN
			xMaskPageBtStart:=FALSE;
		END_IF;
	END_IF;

	(* Set state button start *)
	RisingEdgeSignalStartButton(CLK:=xHWStart);
	IF RisingEdgeSignalStartButton.Q THEN T_StartButton.xInputState:=TRUE; ELSE T_StartButton.xInputState:=FALSE; END_IF
	T_StartButton.xInputState:=T_StartButton.xInputState AND T_VisuQVis.T_ConfigPage[iIndexActivPage].xMaskBtStart;

	(* Led off if action is starting *)
	T_StartButton.xLedState:=T_VisuQVis.T_ConfigPage[iIndexActivPage].xMaskBtStart;

	(* set page mask *)
	T_StartButton.xInputState:=T_StartButton.xInputState AND xMaskPageBtStart;
	T_StartButton.xLedState:=T_StartButton.xLedState AND xMaskPageBtStart;

	T_CtrleBtStartStop.xForceSetStartButton:=FALSE;

(* Stop Button *)
	IF NOT(xNotCheckStateStop) OR T_CtrleBtStartStop.xForceSetStopButton THEN
		IF xProcessActive OR T_CtrleBtStartStop.xForceSetStopButton THEN
			xMaskPageBtStop:=NOT(TProcess.T_Ctrle.xStop) AND (T_ExchgParam.T_Visu.T_Message.iState <> 235);
			IF T_CtrleBtStartStop.xForceSetStopButton THEN
				xMaskPageBtStop:=TRUE;
			END_IF;
			IF (T_ExchgParam.T_Visu.T_Message.iState = 401) THEN
				xMaskPageBtStop:=FALSE;
			END_IF;
		ELSE
			xTmp:=	((((T_ExchgParam.T_Station1.wState AND 16#6) = 16#2)) AND gT_SafetyStatus.xSetupOperateModeActive) OR
					T_VisuQVis.T_CtrleAction.xFunctionActive;
			xTmp:=	xTmp OR
					(((T_VisuQVis.T_CtrleAction.iFunction >= 400) AND (T_VisuQVis.T_CtrleAction.iFunction <= 498)) AND
					NOT(T_VisuQVis.T_CtrleAction.xDone) AND NOT(T_VisuQVis.T_CtrleAction.xErr));
			IF xTmp THEN
				(* Station aktiv *)
				xMaskPageBtStop:=TRUE;
			ELSE
				(* Kein Prozess und keine Stationsfunktion ist aktiv *)
				CASE dwActualPage OF
				gT_PageNumber.iAutoMode_ToolChange:
					IF (T_ExchgParam.T_TeachIn.arAxis[gciAxisZ_St1].bActState AND 16#4) = 16#4 THEN
						xMaskPageBtStop:=TRUE;	(* Achse bewegt sich *)
					END_IF;
				gT_PageNumber.iWorkStation_Axis1:		(* TeachIN für Absolut Bewegung oder Geschwindigkeitsbewegung *)
					CASE T_ExchgParam.T_TeachIn.iSetup_AxisSel OF
					gciAxisZ_St1:
						IF (T_ExchgParam.T_TeachIn.arAxis[gciAxisZ_St1].bActState AND 16#4) = 16#4 THEN
							xMaskPageBtStop:=TRUE;	(* Achse bewegt sich *)
						END_IF;
					gciAxisS_St1,3:
						IF (T_ExchgParam.T_TeachIn.arAxis[gciAxisS_St1].bActState AND 16#4) = 16#4 THEN
							xMaskPageBtStop:=TRUE;	(* Achse bewegt sich *)
						END_IF;
					END_CASE;
				END_CASE;
			END_IF;
		END_IF;
		IF xStationSecurityStateON THEN
			xMaskPageBtStop:=FALSE;
		END_IF;
	END_IF;

	RisingEdgeSignalStopButton(CLK:=xHWStop);
	IF RisingEdgeSignalStopButton.Q THEN T_StopButton.xInputState:=TRUE; ELSE T_StopButton.xInputState:=FALSE; END_IF
	T_StopButton.xInputState:=T_StopButton.xInputState AND T_VisuQVis.T_ConfigPage[iIndexActivPage].xMaskBtStop;

	T_StopButton.xLedState:=T_VisuQVis.T_ConfigPage[iIndexActivPage].xMaskBtStop;

	(* set page mask *)
	T_StopButton.xInputState:=T_StopButton.xInputState AND xMaskPageBtStop;
	T_StopButton.xLedState:=T_StopButton.xLedState AND xMaskPageBtStop;

	T_CtrleBtStartStop.xForceSetStopButton:=FALSE;
END_FUNCTION_BLOCK

(* POU PRG_LAYER4_PROCESS/PRG_PROCESS, FBD *)
PROGRAM PRG_PROCESS
VAR
	FBProcess: FB_PROCESS;
	xReady: BOOL;
	xDone: BOOL;
	xStop: BOOL;
	xReferenced: BOOL;
	xError: BOOL;
	diErrorNr: DINT;
	iFunctionNr: INT;
	FBPreWarningCtrlMessage: FB_PreWarning_Ctrl_Message;
	xEnergyON: BOOL;
END_VAR
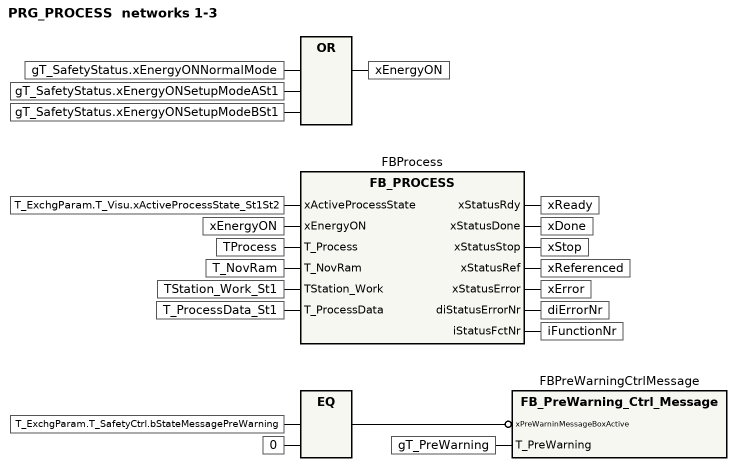
_FBD_ (* Function Block Diagram *)
NETWORK 1
	OR(gT_SafetyStatus.xEnergyONNormalMode, gT_SafetyStatus.xEnergyONSetupModeASt1, gT_SafetyStatus.xEnergyONSetupModeBSt1) => xEnergyON
NETWORK 2
	FBProcess:FB_PROCESS(xActiveProcessState: T_ExchgParam.T_Visu.xActiveProcessState_St1St2, xEnergyON: xEnergyON, T_Process: TProcess, T_NovRam: T_NovRam, TStation_Work: TStation_Work_St1, T_ProcessData: T_ProcessData_St1, xStatusDone => xDone, xStatusStop => xStop, xStatusRef => xReferenced, xStatusError => xError, diStatusErrorNr => diErrorNr, iStatusFctNr => iFunctionNr) => xReady
NETWORK 3
	FBPreWarningCtrlMessage:FB_PreWarning_Ctrl_Message(xPreWarninMessageBoxActive: NOT EQ(T_ExchgParam.T_SafetyCtrl.bStateMessagePreWarning, 0), T_PreWarning: gT_PreWarning)
_END_FBD_
(* the same logic as Structured Text *)
(* Network 1 *)
xEnergyON := gT_SafetyStatus.xEnergyONNormalMode OR gT_SafetyStatus.xEnergyONSetupModeASt1 OR gT_SafetyStatus.xEnergyONSetupModeBSt1;
(* Network 2 *)
FBProcess(xActiveProcessState := T_ExchgParam.T_Visu.xActiveProcessState_St1St2, xEnergyON := xEnergyON, T_Process := TProcess, T_NovRam := T_NovRam, TStation_Work := TStation_Work_St1, T_ProcessData := T_ProcessData_St1);
xDone := FBProcess.xStatusDone;
xStop := FBProcess.xStatusStop;
xReferenced := FBProcess.xStatusRef;
xError := FBProcess.xStatusError;
diErrorNr := FBProcess.diStatusErrorNr;
iFunctionNr := FBProcess.iStatusFctNr;
xReady := FBProcess.xStatusRdy;
(* Network 3 *)
FBPreWarningCtrlMessage(xPreWarninMessageBoxActive := NOT (T_ExchgParam.T_SafetyCtrl.bStateMessagePreWarning = 0), T_PreWarning := gT_PreWarning);
END_PROGRAM

(* POU PRG_LAYER4_PROCESS/FBPROCESS/FB_PROCESS, ST *)
FUNCTION_BLOCK FB_PROCESS
VAR_INPUT
	xActiveProcessState:BOOL;
	xEnergyON:BOOL;
END_VAR
VAR_IN_OUT
	T_Process : ST_PROCESS;
	T_NovRam : ST_NOVRAM;
	TStation_Work : ST_STATION;
	T_ProcessData:ST_PROCESSDATA;
END_VAR
VAR_OUTPUT
	xStatusRdy : BOOL := FALSE;
	xStatusDone : BOOL := FALSE;
	xStatusStop : BOOL := FALSE;
	xStatusRef : BOOL := FALSE;
	xStatusError : BOOL := FALSE;
	diStatusErrorNr : DINT :=0;
	iStatusFctNr : INT := 0;
END_VAR
VAR
	xDisable: BOOL;
	xSetEnd: BOOL;
	RisingEdgeProcessExecute: R_TRIG;
	RisingEdgeProcessStop: R_TRIG;
	RisingEdgeProcessAbord: R_TRIG;
	FBErrorMessage : FB_ErrorMessage;
	xPrcFct_StationError: BOOL;
	xPrcFct_SaveStationError: BOOL;
	iPrcFct_StepStationError: INT;
	xPrcFct_StationReady: BOOL;
	xPrcFct_StationBlock: BOOL;
	xPrcFct_StartMainPrc: BOOL;
	iPrcFct_StepPrc: INT;
	xPrcFct_InitStep: BOOL;
	diPrcFct_SaveErrorNr: DINT;
	xPrcFct_StopProcess: BOOL;
	iPrcFct_StepStopProcess: INT;
	xStartMainPrc: BOOL;
	xPrcFct_StartPrc_Parallel1: BOOL;
	iPrcFct_StepPrc_Parallel1: INT;
	xPrcFct_InitStep_Parallel1: BOOL;
	iPrcFct_StepPrc_Parallel2: INT;
	xPrcFct_InitStep_Parallel2: BOOL;
	xPrcFct_StartPrc_Parallel2: BOOL;
	xPrcFct_SetNextStationActive_St1: BOOL;
	iPrcFct_PickPlaceProcedure: INT;
	TONTickTime: TON;
	FBProcessInformation_StR: FB_ProcessInformation;
	xAutoActiveProcess: BOOL;
	TONTickTime1: TON;
	FBWPCounter_StR: FB_WPCounter;
	xPrcFct_PartDiscReady: BOOL;
	xPrcFct_ReadyToWriteQuality_St1: BOOL;
	xPrcFct_WorkStationReady: BOOL;
	xPrcFct_XAxisGoToWaitPos: BOOL;
	xPrcFct_ForceResetFlag: BOOL;
	xPrcFct_SaveNoMoreParts: BOOL;
	xExecuteOneTime: BOOL;
	ii: INT;
	xHoleToWork: BOOL;
	RisingEdgeCheckWorkEnd: R_TRIG;
	xProcessActive: BOOL;
	xRdyCycleTime: BOOL;
	FBWPAnalysis_StR: FB_WPAnalysis;
	xPrcFct_ProcessContinueActive: BOOL;
	xPrcFct_StopCycleProcess: BOOL;
	xPrcFct_Ready_St1: BOOL;
	xSpindelCalibrationONOFF: BOOL;
	iStepPrc_1: INT;
	xInitPrc_1: BOOL;
	iNumberTryInfeed: INT;
	xActivate_StationRight: BOOL;
	xBlockQuality_StR: BOOL;
	xWriteData: BOOL;
	xStartWorkPart: BOOL;
END_VAR
CtrlInformation;
(******************************************************************************************************************************************)
(***********************************		           Enable/Disable Prozess                           ******************************************)
(******************************************************************************************************************************************)
IF NOT(T_Process.T_Ctrle.xEnable) THEN
	T_Process.T_Ctrle.xRdy:=FALSE;
	xDisable:=TRUE;
	RETURN;
ELSE
	IF xDisable THEN
		T_Process.T_Ctrle.xRdy:=TRUE;
		xDisable:=FALSE;
		xSetEnd:=TRUE;
	END_IF;
END_IF;
CtrlWorkpiece;
(******************************************************************************************************************************************)
(****************************				                  Status Part                                                            *****************************)
(******************************************************************************************************************************************)
xStatusRdy:=T_Process.T_Ctrle.xRdy;
xStatusDone:=T_Process.T_Ctrle.xDone;
xStatusStop:=T_Process.T_Ctrle.xStop;
xStatusRef:=	TStation_Work.TControl.xReferenced;
T_Process.T_Ctrle.xReferenced:=xStatusRef;
xStatusError:=T_Process.T_Ctrle.xError;
diStatusErrorNr:=T_Process.T_Ctrle.diErrorNr;
iStatusFctNr:=T_Process.T_Ctrle.iFunctNr;
(******************************************************************************************************************************************)
(****************************				         Error Controlling Part                                                  *****************************)
(******************************************************************************************************************************************)
CtrlErrorProcess;
(******************************************************************************************************************************************)
(****************************				         Main Controlling Part                                                  *****************************)
(******************************************************************************************************************************************)
CtrlMainProcess;
(******************************************************************************************************************************************)
(****************************				              Funktionen                                                               *****************************)
(******************************************************************************************************************************************)
IF xStartMainPrc AND NOT(xSetEnd) THEN
	IF (T_Process.T_Fct.iFunctNr = 1) THEN
		ProcessFunction_Fct_Referencing;
	END_IF;
	IF (T_Process.T_Fct.iFunctNr = 2) THEN
		ProcessFunction_Fct_Automat;
	END_IF;
	IF (T_Process.T_Fct.iFunctNr = 3) THEN
		ProcessFunction_Fct_HandMode;
		gxHandModeActive:=TRUE;
	ELSE
		gxHandModeActive:=FALSE;
		gxBlockSetQuality:=FALSE;
	END_IF;
ELSE
	gxHandModeActive:=FALSE;
	gxBlockSetQuality:=FALSE;
END_IF;
(******************************************************************************************************************************************)
(****************************				               Init / Reset Flag                                                      *****************************)
(******************************************************************************************************************************************)
IF xSetEnd THEN
	xSetEnd:=FALSE;
	T_Process.T_Ctrle.xStop:=FALSE;
	T_Process.T_Ctrle.xExecute:=FALSE;
	T_Process.T_Ctrle.xDone:=TRUE;
	T_Process.T_Ctrle.xAbordProcess:=FALSE;
	T_Process.T_Ctrle.xError:=FALSE;
	T_Process.T_Ctrle.diErrorNr:=0;
	T_Process.T_Ctrle.xErrorReady:=FALSE;
	T_Process.T_Ctrle.xQuitError:=FALSE;
	T_Process.T_Fct.xSetEndFunction:=TRUE;
	ProcessFunction_Ctrl_End;
	xStartMainPrc:=FALSE;
	xPrcFct_StationBlock:=FALSE;
	iPrcFct_StepStationError:=1;
	xPrcFct_SaveStationError:=FALSE;
	T_Process.T_Fct.xErrorReady:=FALSE;
	TStation_Work.THWWorkStation.TCtrlWork.xActiveProcess:=FALSE;
	TStation_Work.THWWorkStation.TCtrlWork.xWorkingFinished:=FALSE;
	TStation_Work.THWWorkStation.TCtrlWork.xWorkingStarted:=FALSE;
END_IF;
END_FUNCTION_BLOCK
ACTION CtrlErrorProcess:
IF T_Process.T_Fct.xError AND NOT(T_Process.T_Fct.xQuitError) THEN
	(* Bei Fehler wird der Prozess abgebrochen, Bei Warnung kann weitergefahren oder abgebrochen werden *)
	T_Process.T_Ctrle.diErrorNr:=T_Process.T_Fct.diErrorNr;
	T_Process.T_Fct.xQuitError:=TRUE;
END_IF;
IF T_Process.T_Fct.xErrorReady THEN
	IF NOT(T_Process.T_Fct.xQuitError) AND T_Process.T_Fct.xDone AND NOT(T_Process.T_Ctrle.xErrorReady) THEN
		(* Fehler kann nun gesetzt werden *)
		T_Process.T_Ctrle.xError:=TRUE;
		T_Process.T_Ctrle.xErrorReady:=TRUE;
		T_Process.T_Fct.xErrorReady:=FALSE;
	END_IF;
END_IF;
IF T_Process.T_Ctrle.xError THEN
	IF T_Process.T_Ctrle.xQuitError THEN
		T_Process.T_Ctrle.xQuitError:=FALSE;
		IF T_Process.T_Ctrle.xError THEN
			T_Process.T_Ctrle.xError:=FALSE;
			T_Process.T_Ctrle.xErrorReady:=FALSE;
			xSetEnd:=TRUE;
		END_IF;
	END_IF;
END_IF;
END_ACTION
ACTION CtrlInformation:
(* Logik für Wstk Daten Analyse *)
FBWPAnalysis_StR(	diActual_NumberHoleToWork:=  T_NovRam.T_Parameter.T_PartAnalysis[gciStationSt1].diActual_NumberHoleToWork,
					T_PartAnalysis:= T_NovRam.T_Parameter.T_PartAnalysis[gciStationSt1],
					TStation_Work:= TStation_Work,
					xAddInfeedZ:=gxAddInfeedZ,
					xSetPartQuality:=gxSetPartQuality);

(* Prozessinformationen zu den einzelnen Bearbeitungs Stationen *)
FBProcessInformation_StR(	T_Parameter:= T_NovRam.T_Parameter,
							TStation_Work:= TStation_Work);

(* Logik für Automatik Prozesszeit *)
xAutoActiveProcess:=	T_Process.T_Ctrle.xEnable AND
						NOT(T_Process.T_Ctrle.xDone) AND
						NOT(T_Process.T_Ctrle.xError) AND
						(T_Process.T_Ctrle.iFunctNr = 2);

IF xAutoActiveProcess THEN
	TONTickTime(IN:=TRUE,PT:=T#1s);
	IF TONTickTime.Q THEN
		TONTickTime(IN:=FALSE);
		T_NovRam.T_Parameter.T_Machine.T_ParamAutomat.tAutoProcessTime_St1St2:=T_NovRam.T_Parameter.T_Machine.T_ParamAutomat.tAutoProcessTime_St1St2 + T#1s;
		IF T_NovRam.T_Parameter.T_Machine.T_ParamAutomat.tAutoProcessTime_St1St2 >= T#86400s THEN
			IF (T_NovRam.T_Parameter.T_Machine.T_ParamAutomat.iAutoProcessDay_St1St2 < 32767) THEN
				T_NovRam.T_Parameter.T_Machine.T_ParamAutomat.iAutoProcessDay_St1St2:=T_NovRam.T_Parameter.T_Machine.T_ParamAutomat.iAutoProcessDay_St1St2 + 1;
			END_IF;
			T_NovRam.T_Parameter.T_Machine.T_ParamAutomat.tAutoProcessTime_St1St2:=T#0s;
		END_IF;
	END_IF;
ELSE
	TONTickTime(IN:=FALSE);
END_IF;

(* AutoBetrieb Aktiv Zeit-->zeigt die Absolute Zeit von jeder Station wie lange es schon Aktiv ist *)
IF xAutoActiveProcess THEN
	TONTickTime1(IN:=TRUE,PT:=T#0.1s);
	IF TONTickTime1.Q THEN
		TONTickTime1(IN:=FALSE);
		IF TStation_Work.TControl.xEnable AND NOT(TStation_Work.TControl.xDone) AND NOT(TStation_Work.TControl.xError) THEN
			T_NovRam.T_Parameter.T_Machine.T_ParamAutomat.tActualActiveTime_St1:=T_NovRam.T_Parameter.T_Machine.T_ParamAutomat.tActualActiveTime_St1 + T#0.1s;
			IF T_NovRam.T_Parameter.T_Machine.T_ParamAutomat.tActualActiveTime_St1 >= T#86400s THEN
				IF (T_NovRam.T_Parameter.T_Machine.T_ParamAutomat.iActualActiveTime_St1 < 32767) THEN
					T_NovRam.T_Parameter.T_Machine.T_ParamAutomat.iActualActiveTime_St1:=T_NovRam.T_Parameter.T_Machine.T_ParamAutomat.iActualActiveTime_St1 + 1;
				END_IF;
				T_NovRam.T_Parameter.T_Machine.T_ParamAutomat.tActualActiveTime_St1:=T#0s;
			END_IF;
		END_IF;
	END_IF;
ELSE
	TONTickTime1(IN:=FALSE);
END_IF;

(* Wstk Zähler *)
FBWPCounter_StR(	iStationNr:=gciStationSt1,
					T_Parameter:= T_NovRam.T_Parameter,
					T_CtrlWork:= TStation_Work.THWWorkStation.TCtrlWork);
END_ACTION
ACTION CtrlMainProcess:
RisingEdgeProcessExecute(CLK:=T_Process.T_Ctrle.xExecute);
RisingEdgeProcessStop(CLK:=T_Process.T_Ctrle.xStop);
RisingEdgeProcessAbord(CLK:=T_Process.T_Ctrle.xAbordProcess);
(* Prozess Start *)
IF RisingEdgeProcessExecute.Q THEN
	IF T_Process.T_Ctrle.xDone AND NOT(T_Process.T_Ctrle.xError) THEN
		T_Process.T_Ctrle.xStop:=FALSE;
		T_Process.T_Ctrle.xExecute:=FALSE;
		T_Process.T_Ctrle.xDone:=FALSE;
		T_Process.T_Ctrle.xAbordProcess:=FALSE;
		T_Process.T_Ctrle.xError:=FALSE;
		T_Process.T_Ctrle.diErrorNr:=0;
		T_Process.T_Fct.xExecute:=TRUE;
		xStartMainPrc:=TRUE;
		T_Process.T_Fct.iFunctNr:=T_Process.T_Ctrle.iFunctNr;
		xRdyCycleTime:=FALSE;
		xStartWorkPart:=FALSE;
	END_IF;
END_IF;

